	2:	//CleanTip ready?
		IF bStop THEN
			IF fbComplexAction.bBusy THEN
				fbComplexAction.M_Stop();
			ELSE
				nStateAction := 80;
			END_IF
		ELSE
			IF NOT fbComplexAction.bBusy THEN
				A_MoveBack();
				nStateAction := 3;
			END_IF			
		END_IF
		
	3:	//MoveBack
		A_MoveBack();
		IF nStateA_MoveBack >= 80 THEN
			IF nStateA_MoveBack = 99 THEN
				nStateAction := 99;
			ELSE
				nStateAction := 80;
			END_IF
			nStateA_MoveBack := 0;
		END_IF
		
END_CASE
END_ACTION

ACTION A_DilMoveValve:
stError.POUState := nStateAction;

CASE nStateAction OF
	0:	
		IF bStop THEN
			nStateAction := 80;
		ELSE
			IF stGCodeRef.pCurrentTool = 0 THEN
				stError.ErrorId := E_ErrorIdGCode.ERRORID_NoSelectedTool;
				nStateAction := 99;
			ELSE
				IF NOT fbItpReadRParams.bBusy THEN
					MEMSET(ADR(stActionData),0,SIZEOF(stActionData));
					stActionData.eAction := E_Action.ACTION_DilMoveValve;
					stActionData.aParams[1] := LREAL_TO_DINT(alrRParam[1]); //ValvePos
					stError.ErrorId := stGCodeRef.pCurrentTool^.M_ExeAction(stActionData);
					IF stError.ErrorId > 0 THEN
						nStateAction := 99;
					ELSE
						nStateAction := 1;	
					END_IF
				END_IF
			END_IF
		END_IF
		
	1:	//Ready?
		IF bStop THEN
			stGCodeRef.pCurrentTool^.M_CancelAction(E_Action.ACTION_DilMoveValve);
		END_IF
		
		IF NOT stGCodeRef.pCurrentTool^.P_bBusy THEN
			IF stGCodeRef.pCurrentTool^.P_bError THEN
				stError.ErrorId := stGCodeRef.pCurrentTool^.P_nErrorId;
				nStateAction := 99;
			ELSE
				nStateAction := 80;	
			END_IF
		END_IF
END_CASE
END_ACTION

ACTION A_Dispense:
stError.POUState := nStateAction;

CASE nStateAction OF
	0:	//Diluter in Ausgangsposition fahren (BOTTOM)	
		IF bStop THEN
			nStateAction := 80;
		ELSE
			IF stGCodeRef.pCurrentTool = 0 THEN
				stError.ErrorId := E_ErrorIdGCode.ERRORID_NoSelectedTool;
				nStateAction := 99;
			ELSE 
				IF stGCodeRef.pCurrentTool^.P_eObjectType = E_ObjectType.OBJECTTYPE_PassivPip THEN
					pPassivPip := stGCodeRef.pCurrentTool;
				ELSE
					nStateAction := 99;
					RETURN;
				END_IF
				
				IF NOT fbItpReadRParams.bBusy THEN
					MEMSET(ADR(stActionData),0,SIZEOF(stActionData));
					stActionData.eAction := E_Action.ACTION_DilMovePlunger;
					stActionData.aParams[1] := 24000;
					stActionData.aParams[2] := pPassivPip^.P_pDiluter^.P_nConfigReloadSpeed;
					stActionData.aParams[3] := pPassivPip^.P_pDiluter^.P_nValvePosInput;
					stError.ErrorId := pPassivPip^.P_pDiluter^.M_ExeAction(stActionData);
					IF stError.ErrorId > 0 THEN
						nStateAction := 99;
					ELSE
						nStateAction := 1;
					END_IF
				END_IF
			END_IF
		END_IF
		
	1:	//Diluter ready -> Dispensen + Timer für Startbreak starten 
		IF bStop THEN
			pPassivPip^.P_pDiluter^.M_CancelAction(ACTION_DilMovePlunger);
			nStateAction := 80;
		ELSE
			IF NOT pPassivPip^.P_pDiluter^.M_GetActionBusy(ACTION_DilMovePlunger) THEN
				MEMSET(ADR(stActionData),0,SIZEOF(stActionData));
				stActionData.eAction := E_Action.ACTION_Dispense;
				IF alrRParam[1] > 0.0 THEN
					stActionData.aParams[1] := LREAL_TO_DINT(alrRParam[1]); //Quantity
					nStateAction := 3;
				ELSE
					//Es wird mit max. 2 x Spritzen-Volumen dispenst
					stActionData.aParams[1] := pPassivPip^.P_pDiluter^.P_nSyringeSize * 20;
					tDelay := LREAL_TO_TIME(alrRParam[3]);
					IF tDelay > T#0S THEN	//Delay
						timer(IN:=TRUE,PT:=tDelay);	//Timer starten
						stGCodeRef.aToolTable[stGCodeRef.sNciToPlc.Tool].tDelayStart := tDelay;
						nStateAction := 2;
					ELSE
						stGCodeRef.aToolTable[stGCodeRef.sNciToPlc.Tool].tDelayStart := T#0s;
						nStateAction := 80;
					END_IF					
				END_IF
				stActionData.aParams[2] := LREAL_TO_DINT(alrRParam[2]); //Flow
				stError.ErrorId := stGCodeRef.pCurrentTool^.M_ExeAction(stActionData);
				IF stError.ErrorId > 0 THEN
					nStateAction := 99;
				END_IF
			END_IF
		END_IF
		
	2:	//Warten auf Timer
		IF bStop THEN
			timer(IN:= FALSE);
			stGCodeRef.pCurrentTool^.M_CancelAction(E_Action.ACTION_Dispense);
			nStateAction := 80;
			RETURN;
		END_IF
		timer();
		IF timer.Q THEN
			timer(IN:= FALSE);		
			nStateAction := 80;
		END_IF
	
	3:	//Warten bis Dispensen fertig
		IF bStop THEN
			pPassivPip^.M_CancelAction(E_Action.ACTION_Dispense);
			nStateAction := 80;
		ELSE
			IF NOT pPassivPip^.M_GetActionBusy(E_Action.ACTION_Dispense) THEN
				nStateAction := 80;
			END_IF
		END_IF
END_CASE
END_ACTION

ACTION A_DispenseDrops:
stError.POUState := nStateAction;

CASE nStateAction OF
	0:	
		IF bStop THEN
			nStateAction := 80;
		ELSE
			IF stGCodeRef.pCurrentTool = 0 THEN
				stError.ErrorId := E_ErrorIdGCode.ERRORID_NoSelectedTool;
				nStateAction := 99;
			ELSE
				IF NOT fbItpReadRParams.bBusy THEN
					stGCodeRef.aToolTable[stGCodeRef.sNciToPlc.Tool].bIsInAction1 := FALSE;
					MEMSET(ADR(stActionData),0,SIZEOF(stActionData));
					stActionData.eAction := E_Action.ACTION_DispenseDrops;
					stActionData.aParams[1] := LREAL_TO_DINT(alrRParam[1]); //Drops
					stActionData.aParams[2] := 1;
					stActionData.aParams[4] := LREAL_TO_DINT(alrRParam[3]); //Drops für Slave bei TwinPip 
					stError.ErrorId := stGCodeRef.pCurrentTool^.M_ExeAction(stActionData);
					IF stError.ErrorId > 0 THEN
						nStateAction := 99;
					ELSE
						IF stActionData.aParams[1] = 0 THEN //Dauerdispensen
							stGCodeRef.aToolTable[stGCodeRef.sNciToPlc.Tool].bIsInAction1 := TRUE;
							tDelay := LREAL_TO_TIME(alrRParam[2]); //Delay
							IF tDelay > T#0S THEN	//Delay
								timer(IN:=TRUE,PT:=tDelay);	//Timer starten
								stGCodeRef.aToolTable[stGCodeRef.sNciToPlc.Tool].tDelayStart := tDelay;
								nStateAction := 2;								
							ELSE
								stGCodeRef.aToolTable[stGCodeRef.sNciToPlc.Tool].tDelayStart := T#0S;
								nStateAction := 80;
							END_IF
						ELSE
							nStateAction := 1;
						END_IF
					END_IF
				END_IF
			END_IF
		END_IF
		
	1:	//Dispense ready?
		IF bStop THEN
			stGCodeRef.pCurrentTool^.M_CancelAction(E_Action.ACTION_DispenseDrops);
			stGCodeRef.aToolTable[stGCodeRef.sNciToPlc.Tool].bIsInAction1 := FALSE;
		END_IF
		
		IF NOT stGCodeRef.pCurrentTool^.P_bBusy THEN
			stGCodeRef.aToolTable[stGCodeRef.sNciToPlc.Tool].bIsInAction1 := FALSE;
			IF stGCodeRef.pCurrentTool^.P_bError THEN
				stError.ErrorId := stGCodeRef.pCurrentTool^.P_nErrorId;
				nStateAction := 99;
			ELSE
				nStateAction := 80;	
			END_IF
		END_IF
		
	2:	//Warten auf Timer
		IF bStop THEN
			timer(IN:= FALSE);
			stGCodeRef.pCurrentTool^.M_CancelAction(E_Action.ACTION_DispenseDrops);
			stGCodeRef.aToolTable[stGCodeRef.sNciToPlc.Tool].bIsInAction1 := FALSE;
			nStateAction := 80;
			RETURN;
		END_IF
		timer();
		IF timer.Q THEN
			timer(IN:= FALSE);		
			nStateAction := 80;
		END_IF		
END_CASE
END_ACTION

ACTION A_Expose:
stError.POUState := nStateAction;

CASE nStateAction OF
	0:	
		IF bStop THEN
			nStateAction := 80;
		ELSE
			IF stGCodeRef.pCurrentTool = 0 THEN
				stError.ErrorId := E_ErrorIdGCode.ERRORID_NoSelectedTool;
				nStateAction := 99;
			ELSE
				IF NOT fbItpReadRParams.bBusy THEN
					MEMSET(ADR(stActionData),0,SIZEOF(stActionData));
					stActionData.eAction := E_Action.ACTION_Expose;
					stActionData.aParams[1] := LREAL_TO_DINT(alrRParam[1]); //Ctrl
					stActionData.aParams[2] := LREAL_TO_DINT(alrRParam[2]); //Brightness
					stActionData.aParams[3] := LREAL_TO_DINT(alrRParam[3]); //Time
					stError.ErrorId := stGCodeRef.pCurrentTool^.M_ExeAction(stActionData);
					IF stError.ErrorId > 0 THEN
						nStateAction := 99;
					ELSE
						IF stActionData.aParams[3] = 0 THEN
							nStateAction := 80;
						ELSE
							nStateAction := 1;	
						END_IF
					END_IF
				END_IF
			END_IF
		END_IF
		
	1:	//Expose ready?
		IF bStop THEN
			stGCodeRef.pCurrentTool^.M_CancelAction(E_Action.ACTION_Expose);
		END_IF
		
		IF NOT stGCodeRef.pCurrentTool^.P_bBusy THEN
			IF stGCodeRef.pCurrentTool^.P_bError THEN
				stError.ErrorId := stGCodeRef.pCurrentTool^.P_nErrorId;
				nStateAction := 99;
			ELSE
				nStateAction := 80;	
			END_IF
		END_IF
END_CASE
END_ACTION

ACTION A_Extrude:
stError.POUState := nStateAction;
CASE nStateAction OF
	0:	
		IF bStop THEN
			nStateAction := 80;
		ELSE
			IF stGCodeRef.pCurrentTool = 0 THEN
				stError.ErrorId := E_ErrorIdGCode.ERRORID_NoSelectedTool;
				nStateAction := 99;
			ELSE
				IF NOT fbItpReadRParams.bBusy THEN
					//Falls Extruder noch nicht ready, weil er z.B. noch in Decomp-Phase ist, warten!
					IF stGCodeRef.pCurrentTool^.M_GetActionBusy(E_Action.ACTION_Extrude) THEN
						RETURN;
					END_IF
					MEMSET(ADR(stActionData),0,SIZEOF(stActionData));
					stActionData.eAction := E_Action.ACTION_Extrude;
					stActionData.aParams[1] := 0;
					stActionData.aParams[2] := 1; //On
					stError.ErrorId := stGCodeRef.pCurrentTool^.M_ExeAction(stActionData);
					IF stError.ErrorId > 0 THEN
						nStateAction := 99;
					ELSE
						stGCodeRef.aToolTable[stGCodeRef.sNciToPlc.Tool].bIsInAction1 := TRUE;
						tDelay := LREAL_TO_TIME(alrRParam[1]); //Delay (Startbreak)
						IF tDelay > T#0S THEN	//Delay
							timer(IN:=TRUE,PT:=tDelay);	//Timer starten
							stGCodeRef.aToolTable[stGCodeRef.sNciToPlc.Tool].tDelayStart := tDelay;
							nStateAction := 1;								
						ELSE
							stGCodeRef.aToolTable[stGCodeRef.sNciToPlc.Tool].tDelayStart := T#0S;
							nStateAction := 80;
						END_IF
					END_IF
				END_IF
			END_IF
		END_IF
		
	1: //Warten auf Timer
		IF bStop THEN
			timer(IN:= FALSE);
			stGCodeRef.pCurrentTool^.M_CancelAction(E_Action.ACTION_Extrude);
			nStateAction := 80;
			RETURN;
		END_IF
		timer();
		IF timer.Q THEN
			timer(IN:= FALSE);
			nStateAction := 80;
		END_IF
END_CASE
END_ACTION

ACTION A_MeasureTool:
stError.POUState := nStateAction;

IF fbComplexAction.bError THEN
	stError.ErrorId :=fbComplexAction.nErrorId;
	nStateAction := 99;
END_IF

CASE nStateAction OF
	0:	//Aktuelles Tool ausgewählt?
		IF stGCodeRef.pCurrentTool = 0 THEN
			stError.Cmd := E_Action.ACTION_MeasureTool;
			stError.ErrorId := E_ErrorIdGCode.ERRORID_NoSelectedTool;
			nStateAction := 99;
		ELSE
			IF NOT fbItpReadRParams.bBusy THEN
				IF fbObjectDirectory.M_GetObjType(LREAL_TO_UINT(alrRParam[1])) = E_ObjectType.OBJECTTYPE_TipCalibrator THEN
					pTarget := fbObjectDirectory.M_GetObjPointer(LREAL_TO_UINT(alrRParam[1]));
					//NCI-Gruppe auflösen
					fbClearGroup(stGCodeRef:= stGCodeRef, bReGearInSlave:= TRUE, bExecute:= TRUE);
					IF NOT fbClearGroup.bBusy THEN
						IF fbClearGroup.bError THEN
							nStateAction := 99;
							stError.ErrorId := fbClearGroup.nErrorId;
						ELSE
							stCurrentPos := pNewTool^.P_stCurrentPosTotal;
							IF bStop THEN
								nStateAction := 80;
							ELSE
								nStateAction := 1;	
							END_IF
						END_IF
						fbClearGroup(stGCodeRef:= stGCodeRef, bExecute:= FALSE);			
					END_IF
				ELSE
					stError.Cmd := E_Action.ACTION_MeasureTool;
					stError.ObjectId := LREAL_TO_UINT(alrRParam[1]);
					stError.ErrorId := E_ErrorIdCmd.ERRORID_UnsuitableTarget;
					nStateAction := 99;
				END_IF
			END_IF
		END_IF

	1:	//Action "MeasureTool" ausführen
		stMeasToolOldOffset := stGCodeRef.pCurrentTool^.P_stAbsPosTotal;
		MEMSET(ADR(stActionData),0,SIZEOF(stActionData));
		stActionData.eAction := E_Action.ACTION_MeasureTool;
		stActionData.nObject := stGCodeRef.pCurrentTool^.P_nObjectID;
		stActionData.nTarget := pTarget^.P_nObjectID;
		stActionData.aParams[2] := LREAL_TO_DINT(alrRParam[3]);

		stError.ErrorId := fbComplexAction.M_ExeAction(stActionData);
		IF stError.ErrorId > 0 THEN
			nStateAction := 99;
		ELSE
			nStateAction := 2;	
		END_IF
		
	2:	//MeasureTool ready? -> Nullpunkt um neuen Offset verschieben
		IF NOT fbComplexAction.bBusy THEN
			stMeasToolNewOffset := stGCodeRef.pCurrentTool^.P_stAbsPosTotal;
			stGCodeRef.sZeroShiftDesc.fShiftX := stGCodeRef.sZeroShiftDesc.fShiftX + stMeasToolOldOffset.X / 1000 -  stMeasToolNewOffset.X / 1000;
			stGCodeRef.sZeroShiftDesc.fShiftY := stGCodeRef.sZeroShiftDesc.fShiftY + stMeasToolOldOffset.Y / 1000 -  stMeasToolNewOffset.Y / 1000;
			stCurrentPos := stGCodeRef.pCurrentTool^.P_stCurrentPosTotal;
			nStateAction := 3;
		END_IF

	3:	//neuen Offset schreiben
		fbItpWriteZeroShiftEx(bExecute:= TRUE, sNciToPlc:= stGCodeRef.sNciToPlc, nZsNo:= 54, sZeroShiftDesc:= stGCodeRef.sZeroShiftDesc);
		IF NOT fbItpWriteZeroShiftEx.bBusy THEN
			IF fbItpWriteZeroShiftEx.bErr THEN
				stError.ErrorId := UDINT_TO_UINT(fbItpWriteZeroShiftEx.nErrId);
				nStateAction := 99;
			ELSE
				A_MoveBack();
				nStateAction := 4;
			END_IF
			fbItpWriteZeroShiftEx(bExecute:= FALSE, sNciToPlc:= stGCodeRef.sNciToPlc, sZeroShiftDesc:= stGCodeRef.sZeroShiftDesc);
		END_IF
		
	4:	//MoveBack
		A_MoveBack();
		IF nStateA_MoveBack >= 80 THEN
			IF nStateA_MoveBack = 99 THEN
				nStateAction := 99;
			ELSE
				nStateAction := 80;
			END_IF
			nStateA_MoveBack := 0;
		END_IF
END_CASE
END_ACTION

ACTION A_MoveBack:
CASE nStateA_MoveBack OF
	0:	//MoveXY Ausgangspunkt (stCurrentPos)
		MEMSET(ADR(stActionData),0,SIZEOF(stActionData));
		stActionData.eAction := E_Action.ACTION_MoveXY;
		stActionData.aParams[1] := E_MoveMode.MODE_AbsWithOffset;
		stActionData.aParams[2] := REAL_TO_DINT(stCurrentPos.X);
		stActionData.aParams[3] := REAL_TO_DINT(stCurrentPos.Y);
		stActionData.aParams[4] := -1; //max Speed X
		stActionData.aParams[5] := -1; //max Speed Y
		stError.ErrorId := stGCodeRef.pCurrentTool^.M_ExeAction(stActionData);
		IF stError.ErrorId > 0 THEN
			nStateA_MoveBack := 99;
		ELSE
			nStateA_MoveBack := 1;
		END_IF
	
	1:	//MoveXY ready? -> MoveZ Ausgangspunkt (stCurrentPos)
		IF NOT stGCodeRef.pCurrentTool^.M_GetActionBusy(E_Action.ACTION_MoveXY) THEN
			IF stGCodeRef.pCurrentTool^.P_eObjectType = E_ObjectType.OBJECTTYPE_TwinPiezoHolder THEN
				//Einschwenken, falls ausgeschwenkt
				pTwinPiezoHolder := stGCodeRef.pCurrentTool;
				IF pTwinPiezoHolder^.P_eCurrentSwivelState = E_SwivelState.Original THEN
					MEMSET(ADR(stActionData),0,SIZEOF(stActionData));
					stActionData.eAction := E_Action.ACTION_Swivel;
					stActionData.aParams[1] := 1;
					stError.ErrorId := pTwinPiezoHolder^.M_ExeAction(stActionData);
					IF stError.ErrorId > 0 THEN
						nStateA_MoveBack := 99;
					ELSE
						nStateA_MoveBack := 2;
					END_IF
				ELSE
					nStateA_MoveBack := 3;		
				END_IF
			ELSE
				nStateA_MoveBack := 3;	
			END_IF
		END_IF	
	
	2:	//TwinPiezoHolder ready?
		IF NOT stGCodeRef.pCurrentTool^.M_GetActionBusy(E_Action.ACTION_Swivel) THEN
			nStateA_MoveBack := 3;
		END_IF
	
	3:	//NCI-Gruppe wieder erstellen
		fbBuildGroup(stGCodeRef:= stGCodeRef, bExecute:= TRUE);
		IF NOT fbBuildGroup.bBusy THEN
			IF fbBuildGroup.bError THEN
				stError.ErrorId := fbBuildGroup.nErrorId;
				nStateA_MoveBack := 99;
			ELSE
				nStateA_MoveBack := 80;
			END_IF
			fbBuildGroup(stGCodeRef:= stGCodeRef, bExecute:= FALSE);
		END_IF	
END_CASE
END_ACTION

ACTION A_MoveFree:
CASE nStateA_MoveFree OF
	0:	
		MEMSET(ADR(stActionData),0,SIZEOF(stActionData));
		stActionData.eAction := E_Action.ACTION_MoveZ;
		stActionData.aParams[1] := E_MoveMode.MODE_Free;
		stActionData.aParams[3] := -1;

		stError.ErrorId := stGCodeRef.pCurrentTool^.M_ExeAction(stActionData);
		IF stError.ErrorId > 0 THEN
			nStateA_MoveFree := 99;
		ELSE
			nStateA_MoveFree := 1;
		END_IF
	
	1:	//MoveXY ready? -> MoveZ Ausgangspunkt (stCurrentPos)
		IF NOT stGCodeRef.pCurrentTool^.M_GetActionBusy(E_Action.ACTION_MoveZ) THEN
			nStateA_MoveFree := 2;
		END_IF	
	
	2:	//NCI-Gruppe wieder erstellen
		fbBuildGroup(stGCodeRef:= stGCodeRef, bExecute:= TRUE);
		IF NOT fbBuildGroup.bBusy THEN
			IF fbBuildGroup.bError THEN
				stError.ErrorId := fbBuildGroup.nErrorId;
				nStateA_MoveFree := 99;
			ELSE
				nStateA_MoveFree := 80;
			END_IF
			fbBuildGroup(stGCodeRef:= stGCodeRef, bExecute:= FALSE);
		END_IF	
END_CASE
END_ACTION

ACTION A_MoveZHome:
stError.POUState := nStateAction;

IF stGCodeRef.pCurrentTool^.P_bError THEN
	stError.ErrorId := stGCodeRef.pCurrentTool^.P_nErrorId;
	nStateAction := 99;
END_IF

CASE nStateAction OF
	0:	//Aktuelles Tool ausgewählt?
		IF stGCodeRef.pCurrentTool = 0 THEN
			stError.ErrorId := E_ErrorIdGCode.ERRORID_NoSelectedTool;
			nStateAction := 99;
		ELSE //Interpolationsgruppe auflösen (notwendig für Step3)
			fbClearGroup(stGCodeRef:= stGCodeRef,bReGearInSlave:= TRUE, bExecute:= TRUE);
			IF NOT fbClearGroup.bBusy THEN
				IF fbClearGroup.bError THEN
					nStateAction := 99;
					stError.ErrorId := fbClearGroup.nErrorId;
				ELSE
					stCurrentPos := pNewTool^.P_stCurrentPosTotal;
					IF bStop THEN
						nStateAction := 80;
					ELSE
						nStateAction := 1;	
					END_IF
				END_IF
				fbClearGroup(stGCodeRef:= stGCodeRef, bExecute:= FALSE);
			END_IF
		END_IF
		
	1:	//MoveZ
		IF bStop THEN
			nStateAction := 80;
		ELSE
			MEMSET(ADR(stActionData),0,SIZEOF(stActionData));
			stActionData.eAction := E_Action.ACTION_MoveZ;
			stActionData.aParams[1] := E_MoveMode.MODE_Home;
			stActionData.aParams[3]  := -1; //MaxSpeed
			stError.ErrorId := stGCodeRef.pCurrentTool^.M_ExeAction(stActionData);
			IF stError.ErrorId > 0 THEN
				nStateAction := 99;
			ELSE
				nStateAction := 2;
			END_IF
		END_IF
		
	2:	//MoveZ ready? -> aktuelle Position auf Q1-Achse übertragen
		IF NOT stGCodeRef.pCurrentTool^.M_GetActionBusy(E_Action.ACTION_MoveZ) THEN
			stCurrentPos := stGCodeRef.pCurrentTool^.P_stCurrentPosTotal;
 			fbMcSetPosition(Axis:= AxisRefQ1, Execute:= TRUE, Position:= stCurrentPos.Z / 1000.0 - stGCodeRef.sZeroShiftDesc.fShiftZ , Options:= sSetPositionOptions);
			nStateAction := 3;	
		END_IF
		
	3:	//SetPosition ready?
		fbMcSetPosition(Axis:= AxisRefQ1);
		IF NOT fbMcSetPosition.Busy THEN
			IF fbMcSetPosition.Error THEN
				stError.ErrorId := UDINT_TO_UINT(fbMcSetPosition.ErrorID);
				nStateAction := 99;
			ELSE
				IF bStop THEN
					nStateAction := 80;
				ELSE
					nStateAction := 4;	
				END_IF
			END_IF
			fbMcSetPosition(Axis:= AxisRefQ1 , Execute:= FALSE);
		END_IF
		
	4:	//Interpolationsgruppe bilden
		fbBuildGroup(stGCodeRef:= stGCodeRef, bExecute:= TRUE);
		IF NOT fbBuildGroup.bBusy THEN
			IF fbBuildGroup.bError THEN
				stError.ErrorId := fbBuildGroup.nErrorId;
				nStateAction := 99;
			ELSE
				nStateAction := 80;
			END_IF
			fbBuildGroup(stGCodeRef:= stGCodeRef, bExecute:= FALSE);
		END_IF
END_CASE
END_ACTION

ACTION A_PipPostSequence:
stError.POUState := nStateAction;

IF fbComplexAction.bError THEN
	stError.ErrorId :=fbComplexAction.nErrorId;
	nStateAction := 99;
	RETURN;
END_IF

CASE nStateAction OF
	0:	//R-Parameter auswerten und validieren
		IF stGCodeRef.pCurrentTool = 0 THEN
			stError.ErrorId := E_ErrorIdGCode.ERRORID_NoSelectedTool;
			nStateAction := 99;
		ELSE
			IF NOT fbItpReadRParams.bBusy THEN
				//alle Paramter validieren und TargetIds zwischenspeichern
				nTgtNrStrob := LREAL_TO_UINT(alrRParam[1]);
				nDispenseTest := LREAL_TO_DINT(alrRParam[2]);
				
				nTgtNrWS_DispenseWaste1	:= LREAL_TO_UINT(alrRParam[3]);
				nSpecPointNr_DispenseWaste1 := LREAL_TO_UINT(alrRParam[4]);
				nQuantity_DispenseWaste1 := LREAL_TO_DINT(alrRParam[5]);
				nFlow_DispenseWaste1 := LREAL_TO_DINT(alrRParam[6]);
				
				nTgtNrSource := LREAL_TO_UINT(alrRParam[7]);
				nGetSampleColSlotNr := LREAL_TO_DINT(alrRParam[8]);
				nGetSampleRow := LREAL_TO_DINT(alrRParam[9]);
				nGetSampleQuantity := LREAL_TO_DINT(alrRParam[10]);
				nGetSampleFlow := LREAL_TO_DINT(alrRParam[11]);
				nGetSampleDelay := LREAL_TO_DINT(alrRParam[12]);
				
				nTgtNrWS_DispenseWaste2 := LREAL_TO_UINT(alrRParam[13]);
				nSpecPointNr_DispenseWaste2 := LREAL_TO_UINT(alrRParam[14]);
				nQuantity_DispenseWaste2 := LREAL_TO_DINT(alrRParam[15]);
				nFlow_DispenseWaste2 := LREAL_TO_DINT(alrRParam[16]);
				
				nTgtNrWS_Wash1 := LREAL_TO_UINT(alrRParam[17]);
				nSpecPointNr_Wash1 := LREAL_TO_UINT(alrRParam[18]);
				nWashFlow_Wash1 := LREAL_TO_DINT(alrRParam[19]);
				nWashTime_Wash1 := LREAL_TO_DINT(alrRParam[20]);

				nTgtNrWS_Wash2 := LREAL_TO_UINT(alrRParam[21]);
				nSpecPointNr_Wash2 := LREAL_TO_UINT(alrRParam[22]);
				nWashFlow_Wash2 := LREAL_TO_DINT(alrRParam[23]);
				nWashTime_Wash2 := LREAL_TO_DINT(alrRParam[24]);
				
				nTgtNrDryPad_Dry1 := LREAL_TO_UINT(alrRParam[25]);
				nDryCount_Dry1 := LREAL_TO_USINT(alrRParam[26]);
				nDryTime_Dry1 := LREAL_TO_DINT(alrRParam[27]);
				
				//Check 1. DispenseTest
				IF nDispenseTest > 0 THEN
					IF NOT M_ValidateTargetNr(nTgtNrStrob) THEN
						stError.ErrorId := E_ErrorIdGCode.ERRORID_InvalidRParameter;
						stError.ErrorId2 := 1;
						nStateAction := 99;
						RETURN;
					END_IF
				END_IF
				
				//Check 2. DispenseWaste
				IF nQuantity_DispenseWaste1 > 0 THEN
					IF NOT M_ValidateTargetNr(nTgtNrWS_DispenseWaste1) THEN
						stError.ErrorId := E_ErrorIdGCode.ERRORID_InvalidRParameter;
						stError.ErrorId2 := 3;
						nStateAction := 99;
						RETURN;
					END_IF
					//Flow muss größer 0 sein!
				END_IF
				
				//Check 3. GetPipSample (Waschlösung)
				IF nGetSampleQuantity > 0 THEN //wenn 0, dann werden die nächsten beiden Schritte auch ausgelassen und müssen nicht gecheckt werden
					IF M_ValidateTargetNr(nTgtNrSource) THEN
						pTarget := fbObjectDirectory.M_GetObjPointer(stGCodeRef.aTargetTable[nTgtNrSource]);
						IF pTarget = 0 THEN
							stError.ErrorId := E_ErrorIdGCode.ERRORID_InvalidRParameter;
							stError.ErrorId2 := 7;
							nStateAction := 99;
							RETURN;
						END_IF
						IF pTarget^.P_eObjectType = E_ObjectType.OBJECTTYPE_Mtp THEN
							pMtp := pTarget;
							IF NOT(nGetSampleColSlotNr > 0 AND nGetSampleColSlotNr <= pMtp^.P_nCols) THEN
								stError.ErrorId := E_ErrorIdGCode.ERRORID_InvalidRParameter;
								stError.ErrorId2 := 8;
								nStateAction := 99;
								RETURN;
							END_IF
							IF NOT(nGetSampleRow > 0 AND nGetSampleRow <= pMtp^.P_nRows) THEN
								stError.ErrorId := E_ErrorIdGCode.ERRORID_InvalidRParameter;
								stError.ErrorId2 := 9;
								nStateAction := 99;
								RETURN;
							END_IF
						ELSIF pTarget^.P_eObjectType = E_ObjectType.OBJECTTYPE_VialRack THEN
							pVialRack := pTarget;						
							//Im Slot muss auch ein Vial sein!
							pPieceSlot := pVialRack^.M_GetSlot(DINT_TO_UINT(nGetSampleColSlotNr));
							IF pPieceSlot = 0 THEN
								stError.ErrorId := E_ErrorIdGCode.ERRORID_InvalidRParameter;
								stError.ErrorId2 := 8;
								nStateAction := 99;
								RETURN;
							END_IF
							IF pPieceSlot^.P_pPiece = 0 THEN
								stError.ErrorId := E_ErrorIdGCode.ERRORID_InvalidRParameter;
								stError.ErrorId2 := 3;
								nStateAction := 99;
								RETURN;
							END_IF
						END_IF
					ELSE
						stError.ErrorId := E_ErrorIdGCode.ERRORID_InvalidRParameter;
						stError.ErrorId2 := 7;
						nStateAction := 99;
						RETURN;
					END_IF
					
					IF nGetSampleFlow < 1 THEN
						stError.ErrorId := E_ErrorIdGCode.ERRORID_InvalidRParameter;
						stError.ErrorId2 := 11;
						nStateAction := 99;
						RETURN;
					END_IF
					
					//Check 4. DispenseWaste
					IF nQuantity_DispenseWaste2 > 0 THEN
						IF NOT M_ValidateTargetNr(nTgtNrWS_DispenseWaste2) THEN
							stError.ErrorId := E_ErrorIdGCode.ERRORID_InvalidRParameter;
							stError.ErrorId2 := 13;
							nStateAction := 99;
							RETURN;
						END_IF
						
						IF nFlow_DispenseWaste2 = 0 THEN
							stError.ErrorId := E_ErrorIdGCode.ERRORID_InvalidRParameter;
							stError.ErrorId2 := 16;
							nStateAction := 99;
							RETURN;
						END_IF
					END_IF
					//Check 5. WashTool
					IF nWashTime_Wash1 > 0 THEN
						IF NOT M_ValidateTargetNr(nTgtNrWS_Wash1) THEN
							stError.ErrorId := E_ErrorIdGCode.ERRORID_InvalidRParameter;
							stError.ErrorId2 := 17;
							nStateAction := 99;
							RETURN;
						END_IF
						IF nWashFlow_Wash1 = 0 THEN
							stError.ErrorId := E_ErrorIdGCode.ERRORID_InvalidRParameter;
							stError.ErrorId2 := 19;
							nStateAction := 99;
							RETURN;
						END_IF
					END_IF
				END_IF
				
				//Check 6. WashTool
				IF nWashTime_Wash2 > 0 THEN
					IF NOT M_ValidateTargetNr(nTgtNrWS_Wash2) THEN
						stError.ErrorId := E_ErrorIdGCode.ERRORID_InvalidRParameter;
						stError.ErrorId2 := 21;
						nStateAction := 99;
						RETURN;
					END_IF
					IF nWashFlow_Wash2 = 0 THEN
						stError.ErrorId := E_ErrorIdGCode.ERRORID_InvalidRParameter;
						stError.ErrorId2 := 23;
						nStateAction := 99;
						RETURN;
					END_IF
				END_IF
					
				//Check 7. DryPip
				IF nDryCount_Dry1 > 0 THEN
					IF NOT M_ValidateTargetNr(nTgtNrDryPad_Dry1) THEN
						stError.ErrorId := E_ErrorIdGCode.ERRORID_InvalidRParameter;
						stError.ErrorId2 := 25;
						nStateAction := 99;
						RETURN;
					END_IF
				END_IF
				nStateAction := 1;
			END_IF
		END_IF
		
	
	1:	//NCI-Gruppe auflösen
		fbClearGroup(stGCodeRef:= stGCodeRef, bReGearInSlave:= TRUE, bExecute:= TRUE);
		IF NOT fbClearGroup.bBusy THEN
			IF fbClearGroup.bError THEN
				nStateAction := 99;
				stError.ErrorId := fbClearGroup.nErrorId;
			ELSE
				stCurrentPos := pNewTool^.P_stCurrentPosTotal;
				IF bStop THEN
					nStateAction := 80;
				ELSE
					nStateAction := 2;
				END_IF
			END_IF
			fbClearGroup(stGCodeRef:= stGCodeRef, bExecute:= FALSE);			
		END_IF
	
	2:	//DispenseTest start
		IF bStop THEN
			nStateAction := 80;
			RETURN;
		END_IF
		
		IF nDispenseTest > 0 THEN
			MEMSET(ADR(stActionData),0,SIZEOF(stActionData));
			stActionData.eAction := E_Action.ACTION_DispenseTest;
			stActionData.nObject := stGCodeRef.pCurrentTool^.P_nObjectID;
			stActionData.nTarget := stGCodeRef.aTargetTable[nTgtNrStrob];
			stActionData.aParams[1] := nDispenseTest;
			stActionData.aParams[2] := 1; //Inhibit dispense trials
			stError.ErrorId := fbComplexAction.M_ExeAction(stActionData);
			IF stError.ErrorId > 0 THEN
				nStateAction := 99;
			ELSE
				alrRParam[1] := 0.0;
				nStateAction := 3;
			END_IF
		ELSE
			nStateAction := 3;
		END_IF
	
	3:	//DispenseTest ready?
		IF NOT fbComplexAction.bBusy THEN
			IF fbComplexAction.P_bLastActionResult THEN
				alrRParam[1] := DINT_TO_LREAL(fbComplexAction.P_nLastActionResult);
				fbComplexAction.P_bLastActionResult := FALSE;
			END_IF
			//in R-Parameter R140 schreiben
			fbItpWriteRParams(sNciToPlc:= stGCodeRef.sNciToPlc, bExecute:= TRUE, pAddr:= ADR(alrRParam), nIndex:= 140, nCount:= 1);
			IF NOT fbItpWriteRParams.bBusy THEN
				IF fbItpWriteRParams.bErr THEN
					nStateAction := 99;
				ELSE
					nStateAction := 4;
				END_IF
				fbItpWriteRParams(sNciToPlc:= stGCodeRef.sNciToPlc, bExecute:= FALSE);
			END_IF
		END_IF
		
	4:	//DispenseWaste start (WashInside)
		IF bStop THEN
			nStateAction := 80;
			RETURN;
		END_IF
	
		IF nQuantity_DispenseWaste1 > 0 THEN
			MEMSET(ADR(stActionData),0,SIZEOF(stActionData));
			stActionData.eAction := E_Action.ACTION_WashTool;
			stActionData.nObject := stGCodeRef.pCurrentTool^.P_nObjectID;
			stActionData.nTarget := stGCodeRef.aTargetTable[nTgtNrWS_DispenseWaste1];
			stActionData.aParams[1] := nSpecPointNr_DispenseWaste1;
			stActionData.aParams[2] := E_WashMode.MODE_WashInside;
			stActionData.aParams[3] := nQuantity_DispenseWaste1;
			stActionData.aParams[4] := nFlow_DispenseWaste1;
			stError.ErrorId := fbComplexAction.M_ExeAction(stActionData);
			IF stError.ErrorId > 0 THEN
				nStateAction := 99;
			ELSE
				nStateAction := 5;	
			END_IF
		ELSE
			nStateAction := 6;
		END_IF
	
	5:	//DispenseWaste ready?
		IF NOT fbComplexAction.bBusy THEN
			nStateAction := 6;
		END_IF
	
	6:	//GetPipSample start (Waschlösung)
		IF bStop THEN
			nStateAction := 80;
			RETURN;
		END_IF
		IF nGetSampleQuantity > 0 THEN
			MEMSET(ADR(stActionData),0,SIZEOF(stActionData));
			stActionData.eAction := E_Action.ACTION_GetPipSample;
			stActionData.nObject := stGCodeRef.pCurrentTool^.P_nObjectID;
			stActionData.nTarget := stGCodeRef.aTargetTable[nTgtNrSource];
			stActionData.aParams[1] := nGetSampleColSlotNr;
			stActionData.aParams[2] := nGetSampleRow;
			stActionData.aParams[3] := nGetSampleQuantity;
			stActionData.aParams[4] := nGetSampleFlow;
			stActionData.aParams[5] := nGetSampleDelay;
			//stActionData.aParams[6] := nGetSampleAirGap;
			//stActionData.aParams[7] := nGetSampleDilBypass;
			stActionData.aParams[8] := 1; //aktivate Piezo
			stError.ErrorId := fbComplexAction.M_ExeAction(stActionData);
			IF stError.ErrorId > 0 THEN
				nStateAction := 99;
			ELSE
				nStateAction := 7;
			END_IF
		
		ELSE
			nStateAction := 12;
		END_IF

	7:	//GetPipSample ready?
		IF NOT fbComplexAction.bBusy THEN
			nStateAction := 8; //DispenseWaste
		END_IF
	8:	//DispenseWaste start (WashInside)
		IF bStop THEN
			nStateAction := 80;
			RETURN;
		END_IF
		
		IF nQuantity_DispenseWaste2 > 0 THEN
			MEMSET(ADR(stActionData),0,SIZEOF(stActionData));
			stActionData.eAction := E_Action.ACTION_WashTool;
			stActionData.nObject := stGCodeRef.pCurrentTool^.P_nObjectID;
			stActionData.nTarget := stGCodeRef.aTargetTable[nTgtNrWS_DispenseWaste2];
			stActionData.aParams[1] := nSpecPointNr_DispenseWaste2;
			stActionData.aParams[2] := E_WashMode.MODE_WashInside;
			stActionData.aParams[3] := nQuantity_DispenseWaste2;
			stActionData.aParams[4] := nFlow_DispenseWaste2;
			stError.ErrorId := fbComplexAction.M_ExeAction(stActionData);
			IF stError.ErrorId > 0 THEN
				nStateAction := 99;
			ELSE
				nStateAction := 9;
			END_IF
		ELSE
			nStateAction := 10;
		END_IF	
		
	9:	//DispenseWaste ready?
		IF NOT fbComplexAction.bBusy THEN
			nStateAction := 10;
		END_IF
	10:	//WashTool(1) start
		IF bStop THEN
			nStateAction := 80;
			RETURN;
		END_IF
		
		IF nWashTime_Wash1 > 0 THEN
			MEMSET(ADR(stActionData),0,SIZEOF(stActionData));
			stActionData.eAction := E_Action.ACTION_WashTool;
			stActionData.nObject := stGCodeRef.pCurrentTool^.P_nObjectID;
			stActionData.nTarget := stGCodeRef.aTargetTable[nTgtNrWS_Wash1];
			stActionData.aParams[1] := nSpecPointNr_Wash1;
			stActionData.aParams[2] := E_WashMode.MODE_WashInOutside;
			stActionData.aParams[3] := 0; //wenn Quantity 0 dann wird nach Time dispenst?
			stActionData.aParams[4] := nWashFlow_Wash1;
			stActionData.aParams[5] := nWashTime_Wash1;
			stError.ErrorId := fbComplexAction.M_ExeAction(stActionData);
			IF stError.ErrorId > 0 THEN
				nStateAction := 99;
			ELSE
				nStateAction := 11;
			END_IF
		ELSE
			nStateAction := 12;
		END_IF
	11:	//WashTool(1) ready?
		IF NOT fbComplexAction.bBusy THEN
			nStateAction := 12;
		END_IF		

	12:	//WashTool(2) start
		IF bStop THEN
			nStateAction := 80;
			RETURN;
		END_IF
		
		IF nWashTime_Wash2 > 0 THEN
			MEMSET(ADR(stActionData),0,SIZEOF(stActionData));
			stActionData.eAction := E_Action.ACTION_WashTool;
			stActionData.nObject := stGCodeRef.pCurrentTool^.P_nObjectID;
			stActionData.nTarget := stGCodeRef.aTargetTable[nTgtNrWS_Wash2];
			stActionData.aParams[1] := nSpecPointNr_Wash2;
			stActionData.aParams[2] := E_WashMode.MODE_WashInOutside;
			stActionData.aParams[3] := 0; //wenn Quantity 0 dann wird nach Time dispenst?
			stActionData.aParams[4] := nWashFlow_Wash2;
			stActionData.aParams[5] := nWashTime_Wash2;
			stError.ErrorId := fbComplexAction.M_ExeAction(stActionData);
			IF stError.ErrorId > 0 THEN
				nStateAction := 99;
			ELSE
				nStateAction := 13;
			END_IF
		ELSE
			nStateAction := 14;
		END_IF
	13:	//WashTool(2) ready?
		IF NOT fbComplexAction.bBusy THEN
			nStateAction := 14;
		END_IF		
		
	14:	//DryPip
		IF bStop THEN
			nStateAction := 80;
			RETURN;
		END_IF
	
		IF nDryCount_Dry1 > 0 THEN
			MEMSET(ADR(stActionData),0,SIZEOF(stActionData));
			stActionData.eAction := E_Action.ACTION_DryPip;
			stActionData.nObject := stGCodeRef.pCurrentTool^.P_nObjectID;
			stActionData.nTarget := stGCodeRef.aTargetTable[nTgtNrDryPad_Dry1];
			stActionData.aParams[1] := nDryTime_Dry1;
			stError.ErrorId := fbComplexAction.M_ExeAction(stActionData);
			IF stError.ErrorId > 0 THEN
				nStateAction := 99;
			ELSE
				nStateAction := 15;	
			END_IF
		ELSE
			nStateAction := 16;
		END_IF
		
	15:	//DryPip ready?
		IF NOT fbComplexAction.bBusy THEN
			nDryCount_Dry1 := nDryCount_Dry1 - 1;
			IF nDryCount_Dry1 > 0 THEN //wiederholen
				nStateAction := 14;
			ELSE
				nStateAction := 16;
			END_IF
		END_IF
		
	16:	//MoveFree
		A_MoveFree();
		IF nStateA_MoveFree >= 80 THEN
			IF nStateA_MoveFree = 99 THEN
				nStateAction := 99;
			ELSE
				nStateAction := 80;
			END_IF
			nStateA_MoveFree := 0;
		END_IF		
	
END_CASE
END_ACTION

ACTION A_PipPreSequence:
stError.POUState := nStateAction;

IF fbComplexAction.bError THEN
	stError.ErrorId :=fbComplexAction.nErrorId;
	nStateAction := 99;
	RETURN;
END_IF

CASE nStateAction OF
	0:	//R-Parameter auswerten und validieren
		IF stGCodeRef.pCurrentTool = 0 THEN
			stError.ErrorId := E_ErrorIdGCode.ERRORID_NoSelectedTool;
			nStateAction := 99;
		ELSE
			IF NOT fbItpReadRParams.bBusy THEN
				//alle Paramter validieren und TargetIds zwischenspeichern
				nTgtNrWS_Wash1 := LREAL_TO_UINT(alrRParam[1]);
				nSpecPointNr_Wash1 := LREAL_TO_UINT(alrRParam[2]);
				nWashFlow_Wash1 := LREAL_TO_DINT(alrRParam[3]);
				nWashTime_Wash1 := LREAL_TO_DINT(alrRParam[4]);
				nTgtNrDryPad_Dry1 := LREAL_TO_UINT(alrRParam[5]);	//kann auch Washstation mit Airblade sein (ab V2.0.8.9)
				nDryCount_Dry1 := LREAL_TO_USINT(alrRParam[6]);		//bei Washstation ist das der SpecPoint der Airblade
				nDryTime_Dry1 := LREAL_TO_DINT(alrRParam[7]);
				nTgtNrSource := LREAL_TO_UINT(alrRParam[8]);
				nGetSampleColSlotNr := LREAL_TO_DINT(alrRParam[9]);
				nGetSampleRow := LREAL_TO_DINT(alrRParam[10]);
				nGetSampleQuantity := LREAL_TO_DINT(alrRParam[11]);
				nGetSampleFlow := LREAL_TO_DINT(alrRParam[12]);
				nGetSampleDelay := LREAL_TO_DINT(alrRParam[13]);
				nGetSampleAirGap := LREAL_TO_DINT(alrRParam[14]);
				nGetSampleDilBypass := LREAL_TO_DINT(alrRParam[15]);
				nTgtNrDryPad_Dry2 := LREAL_TO_UINT(alrRParam[16]);	//kann auch Washstation mit Airblade sein (ab V2.0.8.9)
				nDryCount_Dry2 := LREAL_TO_USINT(alrRParam[17]);	//bei Washstation ist das der SpecPoint der Airblade
				nDryTime_Dry2 := LREAL_TO_DINT(alrRParam[18]);
				nTgtNrStrob := LREAL_TO_UINT(alrRParam[19]);
				nDispenseTest := LREAL_TO_DINT(alrRParam[20]);
				//Check 1. WashTool
				IF nWashTime_Wash1 > 0 THEN
					IF NOT M_ValidateTargetNr(nTgtNrWS_Wash1) THEN
						stError.ErrorId := E_ErrorIdGCode.ERRORID_InvalidRParameter;
						stError.ErrorId2 := 1;
						nStateAction := 99;
						RETURN;
					END_IF
				END_IF
				//Check 2. DryPip
				IF nDryCount_Dry1 > 0 THEN
					IF NOT M_ValidateTargetNr(nTgtNrDryPad_Dry1) THEN
						stError.ErrorId := E_ErrorIdGCode.ERRORID_InvalidRParameter;
						stError.ErrorId2 := 5;
						nStateAction := 99;
						RETURN;
					END_IF
				END_IF
				//Check 3. GetPipSample
				IF nGetSampleQuantity  > 0 THEN
					IF M_ValidateTargetNr(nTgtNrSource) THEN
						pTarget := fbObjectDirectory.M_GetObjPointer(stGCodeRef.aTargetTable[nTgtNrSource]);
						IF pTarget = 0 THEN
							stError.ErrorId := E_ErrorIdGCode.ERRORID_InvalidRParameter;
							stError.ErrorId2 := 8;
							nStateAction := 99;
							RETURN;
						END_IF
						IF pTarget^.P_eObjectType = E_ObjectType.OBJECTTYPE_Mtp THEN
							pMtp := pTarget;
							IF NOT(nGetSampleColSlotNr > 0 AND nGetSampleColSlotNr <= pMtp^.P_nCols) THEN
								stError.ErrorId := E_ErrorIdGCode.ERRORID_InvalidRParameter;
								stError.ErrorId2 := 9;
								nStateAction := 99;
								RETURN;
							END_IF
							IF NOT(nGetSampleRow > 0 AND nGetSampleRow <= pMtp^.P_nRows) THEN
								stError.ErrorId := E_ErrorIdGCode.ERRORID_InvalidRParameter;
								stError.ErrorId2 := 10;
								nStateAction := 99;
								RETURN;
							END_IF
						ELSIF pTarget^.P_eObjectType = E_ObjectType.OBJECTTYPE_VialRack THEN
							pVialRack := pTarget;						
							//Im Slot muss auch ein Vial sein!
							pPieceSlot := pVialRack^.M_GetSlot(DINT_TO_UINT(nGetSampleColSlotNr));
							IF pPieceSlot = 0 THEN
								stError.ErrorId := E_ErrorIdGCode.ERRORID_InvalidRParameter;
								stError.ErrorId2 := 9;
								nStateAction := 99;
								RETURN;
							END_IF
							IF pPieceSlot^.P_pPiece = 0 THEN
								stError.ErrorId := E_ErrorIdGCode.ERRORID_InvalidRParameter;
								stError.ErrorId2 := 9;
								nStateAction := 99;
								RETURN;
							END_IF
						END_IF
					ELSE
						stError.ErrorId := E_ErrorIdGCode.ERRORID_InvalidRParameter;
						stError.ErrorId2 := 8;
						nStateAction := 99;
						RETURN;
					END_IF
					
					IF nGetSampleFlow < 1 THEN
						stError.ErrorId := E_ErrorIdGCode.ERRORID_InvalidRParameter;
						stError.ErrorId2 := 12;
						nStateAction := 99;
						RETURN;
					END_IF
					
					//Check 4. DryPip
					IF nDryCount_Dry2 > 0 THEN
						IF NOT M_ValidateTargetNr(nTgtNrDryPad_Dry2) THEN
							stError.ErrorId := E_ErrorIdGCode.ERRORID_InvalidRParameter;
							stError.ErrorId2 := 16;
							nStateAction := 99;
							RETURN;
						END_IF
					END_IF
					
					IF nDispenseTest > 0 AND NOT M_ValidateTargetNr(nTgtNrStrob) THEN
						stError.ErrorId := E_ErrorIdGCode.ERRORID_InvalidRParameter;
						stError.ErrorId2 := 18;
						nStateAction := 99;
						RETURN;
					END_IF
					
				END_IF
				nStateAction := 1;
			END_IF
		END_IF
		
	1:	//NCI-Gruppe auflösen
		fbClearGroup(stGCodeRef:= stGCodeRef, bReGearInSlave:= TRUE, bExecute:= TRUE);
		IF NOT fbClearGroup.bBusy THEN
			IF fbClearGroup.bError THEN
				nStateAction := 99;
				stError.ErrorId := fbClearGroup.nErrorId;
			ELSE
				stCurrentPos := pNewTool^.P_stCurrentPosTotal;
				IF bStop THEN
					nStateAction := 80;
				ELSE
					nStateAction := 2;
				END_IF
			END_IF
			fbClearGroup(stGCodeRef:= stGCodeRef, bExecute:= FALSE);			
		END_IF
		
	2:	//1. WashTool start
		IF bStop THEN
			nStateAction := 80;
			RETURN;
		END_IF
		
		IF nWashTime_Wash1 > 0 THEN
			MEMSET(ADR(stActionData),0,SIZEOF(stActionData));
			stActionData.eAction := E_Action.ACTION_WashTool;
			stActionData.nObject := stGCodeRef.pCurrentTool^.P_nObjectID;
			stActionData.nTarget := stGCodeRef.aTargetTable[nTgtNrWS_Wash1];
			stActionData.aParams[1] := nSpecPointNr_Wash1;
			stActionData.aParams[2] := E_WashMode.MODE_WashInOutside;
			stActionData.aParams[3] := 0; //wenn Quantity 0 dann wird nach Time dispenst?
			stActionData.aParams[4] := nWashFlow_Wash1;
			stActionData.aParams[5] := nWashTime_Wash1;
			stError.ErrorId := fbComplexAction.M_ExeAction(stActionData);
			IF stError.ErrorId > 0 THEN
				nStateAction := 99;
			ELSE
				nStateAction := 3;	
			END_IF
		ELSE
			nStateAction := 4;
		END_IF
		
	3:	//1. WashTool ready?
		IF NOT fbComplexAction.bBusy THEN
			nStateAction := 4;
		END_IF
		
	4:	//2. DryPip start
		IF bStop THEN
			nStateAction := 80;
			RETURN;
		END_IF
	
		//Ab V2.0.8.9 wird unterschieden, ob auf Drypad oder Washstation mit Airblade getrockent wird.
		IF nDryCount_Dry1 > 0 THEN
			MEMSET(ADR(stActionData),0,SIZEOF(stActionData));
			stActionData.nObject := stGCodeRef.pCurrentTool^.P_nObjectID;
			stActionData.nTarget := stGCodeRef.aTargetTable[nTgtNrDryPad_Dry1];
			
			pTarget := fbObjectDirectory.M_GetObjPointer(stGCodeRef.aTargetTable[nTgtNrDryPad_Dry1]);
			IF pTarget^.P_eObjectType = E_ObjectType.OBJECTTYPE_DryPad THEN
				stActionData.eAction := E_Action.ACTION_DryPip;
				stActionData.aParams[1] := nDryTime_Dry1;
			ELSIF pTarget^.P_eObjectType = E_ObjectType.OBJECTTYPE_WashStation THEN
				stActionData.eAction := E_Action.ACTION_WashTool;
				stActionData.aParams[1] := nDryCount_Dry1; //Specpoint
				stActionData.aParams[2] := E_WashMode.MODE_DryOutside;
				stActionData.aParams[5] := nDryTime_Dry1;
			ELSE
				stError.ErrorId := E_ErrorIdCmd.ERRORID_InvalidTarget;
			END_IF
			
			IF stError.ErrorId > 0 THEN
				nStateAction := 99;
			ELSE
				stError.ErrorId := fbComplexAction.M_ExeAction(stActionData);
				IF stError.ErrorId > 0 THEN
					nStateAction := 99;
				ELSE
					nStateAction := 5;	
				END_IF
			END_IF
		ELSE
			nStateAction := 6; //GetPipSample	
		END_IF
	
	5:	//2. DryPip ready?
		IF NOT fbComplexAction.bBusy THEN
			IF pTarget^.P_eObjectType = E_ObjectType.OBJECTTYPE_DryPad THEN
				nDryCount_Dry1 := nDryCount_Dry1 - 1;
				IF nDryCount_Dry1 > 0 THEN
					nStateAction := 4;
				ELSE
					nStateAction := 6; //GetSample
				END_IF
			ELSE
				nStateAction := 6; //GetSample
			END_IF
		END_IF
		
	6:	//3. GetSample start
		IF bStop THEN
			nStateAction := 80;
			RETURN;
		END_IF
	
		IF nGetSampleQuantity > 0 THEN
			MEMSET(ADR(stActionData),0,SIZEOF(stActionData));
			stActionData.eAction := E_Action.ACTION_GetPipSample;
			stActionData.nObject := stGCodeRef.pCurrentTool^.P_nObjectID;
			stActionData.nTarget := stGCodeRef.aTargetTable[nTgtNrSource];
			stActionData.aParams[1] := nGetSampleColSlotNr;
			stActionData.aParams[2] := nGetSampleRow;
			stActionData.aParams[3] := nGetSampleQuantity;
			stActionData.aParams[4] := nGetSampleFlow;
			stActionData.aParams[5] := nGetSampleDelay;
			stActionData.aParams[6] := nGetSampleAirGap;
			stActionData.aParams[7] := nGetSampleDilBypass;
			stError.ErrorId := fbComplexAction.M_ExeAction(stActionData);
			IF stError.ErrorId > 0 THEN
				nStateAction := 99;
			ELSE
				nStateAction := 7;
			END_IF
		ELSE
			nStateAction := 8; //DryPip zum Zweiten
		END_IF
	
	7:	//3. GetSample ready?
		IF NOT fbComplexAction.bBusy THEN
			nStateAction := 8; //DryPip zum Zweiten
		END_IF
		
	8:	//4. DryPip start
		IF bStop THEN
			nStateAction := 80;
			RETURN;
		END_IF
	
		IF nDryCount_Dry2 > 0 THEN
			MEMSET(ADR(stActionData),0,SIZEOF(stActionData));
			stActionData.nObject := stGCodeRef.pCurrentTool^.P_nObjectID;
			stActionData.nTarget := stGCodeRef.aTargetTable[nTgtNrDryPad_Dry2];
			
			pTarget := fbObjectDirectory.M_GetObjPointer(stGCodeRef.aTargetTable[nTgtNrDryPad_Dry2]);
			IF pTarget^.P_eObjectType = E_ObjectType.OBJECTTYPE_DryPad THEN
				stActionData.eAction := E_Action.ACTION_DryPip;
				stActionData.aParams[1] := nDryTime_Dry2;
			ELSIF pTarget^.P_eObjectType = E_ObjectType.OBJECTTYPE_WashStation THEN
				stActionData.eAction := E_Action.ACTION_WashTool;
				stActionData.aParams[1] := nDryCount_Dry2; //Specpoint
				stActionData.aParams[2] := E_WashMode.MODE_DryOutside;
				stActionData.aParams[5] := nDryTime_Dry2;
			ELSE
				stError.ErrorId := E_ErrorIdCmd.ERRORID_InvalidTarget;
			END_IF
			
			IF stError.ErrorId > 0 THEN
				nStateAction := 99;
			ELSE
				stError.ErrorId := fbComplexAction.M_ExeAction(stActionData);
				IF stError.ErrorId > 0 THEN
					nStateAction := 99;
				ELSE
					nStateAction := 9;
				END_IF
			END_IF
		ELSE
			IF nDispenseTest > 0 THEN
				nStateAction := 10; //DispenseTest
			ELSE
				nStateAction := 12;
			END_IF
		END_IF
	
	9:	//DryPip ready?
		IF NOT fbComplexAction.bBusy THEN
			IF pTarget^.P_eObjectType = E_ObjectType.OBJECTTYPE_DryPad THEN
				nDryCount_Dry2 := nDryCount_Dry2 - 1;
				IF nDryCount_Dry2 > 0 THEN //wiederholen
					nStateAction := 8;
				ELSE
					IF nDispenseTest > 0 THEN
						nStateAction := 10; //DispenseTest
					ELSE
						nStateAction := 12;
					END_IF
				END_IF
			ELSE
				IF nDispenseTest > 0 THEN
					nStateAction := 10; //DispenseTest
				ELSE
					nStateAction := 12;
				END_IF
			END_IF
		END_IF
		
	10:	//DispenseTest start
		IF bStop THEN
			nStateAction := 80;
			RETURN;
		END_IF
	
		MEMSET(ADR(stActionData),0,SIZEOF(stActionData));
		stActionData.eAction := E_Action.ACTION_DispenseTest;
		stActionData.nObject := stGCodeRef.pCurrentTool^.P_nObjectID;
		stActionData.nTarget := stGCodeRef.aTargetTable[nTgtNrStrob];
		stActionData.aParams[1] := nDispenseTest;
		fbComplexAction.P_nDispenseTrials := 0;
		stError.ErrorId := fbComplexAction.M_ExeAction(stActionData);
		IF stError.ErrorId > 0 THEN
			nStateAction := 99;
		ELSE
			alrRParam[1] := 0.0;
			nStateAction := 11;
		END_IF
	
	11:	//DispenseTest ready?
		IF NOT fbComplexAction.bBusy THEN
			IF fbComplexAction.P_bLastActionResult THEN
				alrRParam[1] := DINT_TO_LREAL(fbComplexAction.P_nLastActionResult);
				fbComplexAction.P_bLastActionResult := FALSE;
			END_IF
			//in R-Parameter R140 schreiben
			fbItpWriteRParams(sNciToPlc:= stGCodeRef.sNciToPlc, bExecute:= TRUE, pAddr:= ADR(alrRParam), nIndex:= 140, nCount:= 1);
			IF NOT fbItpWriteRParams.bBusy THEN
				IF fbItpWriteRParams.bErr THEN
					nStateAction := 99;
				ELSE
					nStateAction := 12;	
				END_IF
				fbItpWriteRParams(sNciToPlc:= stGCodeRef.sNciToPlc, bExecute:= FALSE);
			END_IF
		END_IF
		
	12:	//MoveFree
		A_MoveFree();
		IF nStateA_MoveFree >= 80 THEN
			IF nStateA_MoveFree = 99 THEN
				nStateAction := 99;
			ELSE
				nStateAction := 80;
			END_IF
			nStateA_MoveFree := 0;
		END_IF	
END_CASE
END_ACTION

ACTION A_SelectTool:
//+++++++++++++++++++++++++++++++++++++++++++++++++++++++++++++++++++++++++++++++++++++++++++++++++++++++++++++
//Änderung ab V2.0.17!
//Beim Toolwechsel wird nicht mehr der Druck oder der Feed eingestellt.
//Nach einem Toolwechsel sollte daher immer M102 ausgeführt werden
stError.POUState := nStateAction;

CASE nStateAction OF
	0:	
		IF bStop THEN
			nStateAction := 80;
		ELSE
			//Checken, ob Toolnummer (T-Paramter) gültig
			IF NOT (stGCodeRef.sNciToPlc.Tool > 0 AND stGCodeRef.sNciToPlc.Tool <= GCode.cMaxGCodeTools) THEN
				stError.ErrorId := E_ErrorIdGCode.ERRORID_InvalidToolNr;
				nStateAction := 99;
				RETURN;
			ELSE
				//Checken, ob ein gültiges Werkzeug zugeordnet
				IF stGCodeRef.aToolTable[stGCodeRef.sNciToPlc.Tool].pMzTool = 0 OR 
											NOT stGCodeRef.aToolTable[stGCodeRef.sNciToPlc.Tool].bIsUsed THEN
					stError.ErrorId := E_ErrorIdGCode.ERRORID_InvalidToolNr;
					nStateAction := 99;
					RETURN;
				END_IF
			END_IF
			
			pNewTool := stGCodeRef.aToolTable[stGCodeRef.sNciToPlc.Tool].pMzTool;
			
			//Achsen freifahren
			IF pNewTool^.P_bIsMESTool THEN //MES-Tool wird vom Freifahren ausgeschlossen, da Faden abreißen würde
				stError.ErrorId := stGCodeRef.pHead^.M_MoveFree(pNewTool);
			ELSE
				stError.ErrorId := stGCodeRef.pHead^.M_MoveFree(0);	
			END_IF
			
			IF stError.ErrorId > 0 THEN
				nStateAction := 99;
				RETURN;
			END_IF
			nStateAction := 1;
		END_IF
		
	1:	//Achsen ready?
		IF NOT stGCodeRef.pHead^.M_GetActionBusy(E_Action.ACTION_MoveZ) THEN
			nStateAction := 3;
			IF bStop THEN
				nStateAction := 80;
			ELSE
				IF pNewTool^.P_eObjectType = E_ObjectType.OBJECTTYPE_TwinPiezoHolder THEN
					pTwinPiezoHolder := pNewTool;
					IF pTwinPiezoHolder^.P_eCurrentSwivelState <> E_SwivelState.Swiveled THEN
						//Einschwenken
						MEMSET(ADR(stActionData),0,SIZEOF(stActionData));
						stActionData.eAction := E_Action.ACTION_Swivel;
						stActionData.aParams[1] := 1;
						stError.ErrorId := pTwinPiezoHolder^.M_ExeAction(stActionData);
						IF stError.ErrorId > 0 THEN
							nStateAction := 99;
							RETURN;					
						END_IF
						nStateAction := 2;	//warten bis eingeschwenkt
					END_IF
 				END_IF
			END_IF
		END_IF
		
		IF stGCodeRef.pHead^.P_bError THEN
			stError.ErrorId := stGCodeRef.pHead^.P_nErrorId;
			nStateAction := 99;
			RETURN;
		END_IF
	
	2:	//TwinPiezoHolder eingeschwenkt?
		IF bStop THEN
			pNewTool^.M_CancelAction(E_Action.ACTION_Swivel);
			nStateAction := 80;
			RETURN;
		END_IF
		
		IF NOT pNewTool^.M_GetActionBusy(E_Action.ACTION_Swivel) THEN
			nStateAction := 3;
		END_IF
		

		//hier kommt dann noch ein zusätzlicher Offset hinzu, welcher sich aus der zukünftigen Objektvermessung ergibt
	3:	//Neue Nullpunktverschiebeung berechnen (Offset vom aktuellen mit Offset von neuem Tool verrechnen)
		//Es gibt 2 Fälle
		IF stGCodeRef.pCurrentTool = 0 THEN //Es erfolgt die erstmalige Tool-auswahl
			stPos1 := stGCodeRef.pHead^.P_stAbsPosTotal;
		ELSE //Es wurde bereits ein Tool ausgewählt -> es findet ein Toolwechsel statt
			stPos1 := stGCodeRef.pCurrentTool^.P_stAbsPosTotal;
		END_IF
			
		stPos2 := pNewTool^.P_stAbsPosTotal;
		
		stGCodeRef.sZeroShiftDesc.fShiftX := stGCodeRef.sZeroShiftDesc.fShiftX + stPos1.X / 1000.0 -  stPos2.X / 1000.0;
		stGCodeRef.sZeroShiftDesc.fShiftY := stGCodeRef.sZeroShiftDesc.fShiftY + stPos1.Y / 1000.0 -  stPos2.Y / 1000.0;

		stGCodeRef.pCurrentTool := pNewTool;
		
		nStateAction := 4;
	
	4:	//Neue Nullpunktverschiebung schreiben
		fbItpWriteZeroShiftEx(bExecute:= TRUE, sNciToPlc:= stGCodeRef.sNciToPlc, nZsNo:= 54, sZeroShiftDesc:= stGCodeRef.sZeroShiftDesc);	
 		IF NOT fbItpWriteZeroShiftEx.bBusy THEN
			IF fbItpWriteZeroShiftEx.bErr THEN
				nStateAction := 99;
			ELSE
				IF bStop THEN
					nStateAction := 80;
				ELSE
					nStateAction := 5;
				END_IF
			END_IF
			fbItpWriteZeroShiftEx(bExecute:= FALSE, sNciToPlc:= stGCodeRef.sNciToPlc, nZsNo:= 54, sZeroShiftDesc:= stGCodeRef.sZeroShiftDesc);
		END_IF
		
	5:	//NCI-Gruppe auflösen
		fbClearGroup(stGCodeRef:= stGCodeRef, bReGearInSlave:= TRUE, bExecute:= TRUE);
		IF NOT fbClearGroup.bBusy THEN
			IF fbClearGroup.bError THEN
				nStateAction := 99;
				stError.ErrorId := fbClearGroup.nErrorId;
			ELSE
				stCurrentPos := pNewTool^.P_stCurrentPosTotal;
				IF bStop THEN
					nStateAction := 80;
				ELSE
					nStateAction := 6;
				END_IF
				
			END_IF
			fbClearGroup(stGCodeRef:= stGCodeRef, bExecute:= FALSE);
		END_IF
		
	6:	//die aktuelle Position des Tools auf die Q1-Achse übertragen
		fbMcSetPosition(Axis:= AxisRefQ1 , Execute:= TRUE, Position:= stCurrentPos.Z / 1000.0 - stGCodeRef.sZeroShiftDesc.fShiftZ , Options:= sSetPositionOptions);
		IF NOT fbMcSetPosition.Busy THEN
			IF fbMcSetPosition.Error THEN
				nStateAction := 99;
			ELSE
				IF bStop THEN
					nStateAction := 80;
				ELSE
					nStateAction := 7;
				END_IF
			END_IF
			fbMcSetPosition(Axis:= AxisRefQ1 , Execute:= FALSE);
		END_IF
		
	7:	//NCI-Gruppe wieder erstellen
		fbBuildGroup(stGCodeRef:= stGCodeRef, bExecute:= TRUE);
		IF NOT fbBuildGroup.bBusy THEN
			IF fbBuildGroup.bError THEN
				stError.ErrorId := fbBuildGroup.nErrorId;
				nStateAction := 99;
			ELSE
				nStateAction := 80;
			END_IF
			fbBuildGroup(stGCodeRef:= stGCodeRef, bExecute:= FALSE);
		END_IF
END_CASE
END_ACTION

ACTION A_Sequence:
stError.POUState := nStateAction;

IF fbComplexAction.bError THEN
	stError.ErrorId :=fbComplexAction.nErrorId;
	nStateAction := 99;
END_IF

IF nStateAction = 0 THEN
	IF stGCodeRef.pCurrentTool = 0 THEN
		//stError.Cmd := E_Action.ACTION_;;
		stError.ErrorId := E_ErrorIdGCode.ERRORID_NoSelectedTool;
		nStateAction := 99;
	ELSE
		IF NOT fbItpReadRParams.bBusy THEN
			nSequenceNr := LREAL_TO_UINT(alrRParam[1]);
			//SequenceNr 1..5 ?
			IF nSequenceNr >= 1 AND nSequenceNr <= 5 THEN
				pSequence := fbSequenceList.M_Get(stGCodeRef.aSequenceIds[nSequenceNr]);
				//Gültige SubSequence?
				IF pSequence > 0 THEN
					//Sequence schon busy?
					IF NOT((pSequence^.eCurrentState = E_SequenceState.State_Idle) OR (pSequence^.eCurrentState = E_SequenceState.State_Ready)) THEN
						nStateAction := 99;
						stError.ErrorId := E_ErrorIdGCode.ERRORID_InvalidSequenceNr;
						RETURN;
					END_IF
					//Steps vorhanden?
					stError.ErrorId := pSequence^.M_CheckForStart();
					IF stError.ErrorId = 0 THEN
						//NCI-Gruppe auflösen
						fbClearGroup(stGCodeRef:= stGCodeRef, bReGearInSlave:= TRUE, bExecute:= TRUE);
						IF NOT fbClearGroup.bBusy THEN
							IF fbClearGroup.bError THEN
								nStateAction := 99;
								stError.ErrorId := fbClearGroup.nErrorId;
							ELSE
								stCurrentPos := pNewTool^.P_stCurrentPosTotal;
								IF bStop THEN
									nStateAction := 80;
								ELSIF bPause THEN
									nStateAction := 2; //sofort in Pause gehen
								ELSE
									GCode.P_bMoveActionsLocked := FALSE;
									pSequence^.M_Start(0);									
									nStateAction := 3; //perform sequence
								END_IF
							END_IF
							fbClearGroup(stGCodeRef:= stGCodeRef, bExecute:= FALSE);			
						END_IF
					ELSE
						nStateAction := 99;				
					END_IF
				ELSE
					stError.ErrorId := E_ErrorIdCmd.ERRORID_SequenceNotExists;
					nStateAction := 99;
				END_IF				
			ELSE
				stError.ErrorId := E_ErrorIdGCode.ERRORID_InvalidSequenceNr;
				nStateAction := 99;
			END_IF
		END_IF
	END_IF
END_IF

IF nStateAction = 1 THEN //Sequence pausieren
	pSequence^.M_Pause();
	pSequence^();
	IF pSequence^.eCurrentState = E_SequenceState.State_Pause THEN
		nStateAction := 2;
	ELSIF pSequence^.eCurrentState = E_SequenceState.State_Error THEN
		nStateAction := 99;
	ELSIF pSequence^.eCurrentState = E_SequenceState.State_Ready THEN
		pSequence^.M_Reset();
		nStateAction := 80;
		RETURN;
	END_IF
ELSIF nStateAction = 2 THEN //Sequence ist pausiert
	IF bStop THEN
		pSequence^.M_Stop();
		nStateAction := 3;
	ELSIF bPause THEN
		bIsInPause := TRUE;
		RETURN;
	ELSIF bContinue THEN
		IF pSequence^.eCurrentState = E_SequenceState.State_Pause THEN	
			pSequence^.M_Continue();
		ELSIF pSequence^.eCurrentState = E_SequenceState.State_Idle THEN //wurde noch nicht gestartet
			pSequence^.M_Start(0);
		END_IF
		nStateAction := 3;
	END_IF
END_IF

IF nStateAction = 3 THEN //perform sequence , wait for ready
	bIsInPause := FALSE;
	IF bStop THEN
		pSequence^.M_Stop();
	ELSIF bPause THEN
		pSequence^.M_Pause();
		nStateAction := 1;
	END_IF
	pSequence^();
	IF pSequence^.eCurrentState = E_SequenceState.State_Ready THEN
		pSequence^.M_Reset();
		nStateAction := 4;
		GCode.P_bMoveActionsLocked := TRUE;
	ELSIF pSequence^.eCurrentState = E_SequenceState.State_Canceled THEN
		pSequence^.M_Reset();
		nStateAction := 80;
	ELSIF pSequence^.eCurrentState = E_SequenceState.State_Error THEN
		pSequence^.M_Reset();
		nStateAction := 99;
	END_IF
END_IF

IF nStateAction = 4 THEN //MoveBack
	A_MoveBack();
	IF nStateA_MoveBack >= 80 THEN
		IF nStateA_MoveBack = 99 THEN
			nStateAction := 99;
		ELSE
			nStateAction := 80;
		END_IF
		nStateA_MoveBack := 0;
	END_IF	
END_IF
END_ACTION

ACTION A_SetPrintParams:
stError.POUState := nStateAction;

IF nStateAction = 0 THEN
	IF NOT fbItpReadRParams.bBusy THEN
		nToolNr := LREAL_TO_USINT(alrRParam[1]);
		ePrintParamType := LREAL_TO_USINT(alrRParam[2]);
		nPrintParamNumerator := LREAL_TO_USINT(alrRParam[3]);
		nPrintParamValue := LREAL_TO_DINT(alrRParam[4]);
		IF nToolNr = 0 THEN //ausgewähltes Tool benutzen
			pNewTool := stGCodeRef.pCurrentTool;
		ELSIF nToolNr >= 1 AND nToolNr <= GCode.cMaxGCodeTools THEN
			pNewTool := stGCodeRef.aToolTable[nToolNr].pMzTool;
		END_IF
		nStateAction := 1;
		IF pNewTool = 0 THEN
			stError.ErrorId := E_ErrorIdGCode.ERRORID_InvalidToolNr;
			nStateAction := 99;
		END_IF
	END_IF
END_IF

IF nStateAction = 1 THEN
	stMethResult := pNewTool^.M_SetPrintParams(ePrintParamType, nPrintParamNumerator, nPrintParamValue);
	IF NOT stMethResult.bBusy THEN
		IF stMethResult.bError THEN
			stError.ObjectId := pNewTool^.P_nObjectID;
			stError.ErrorId := nErrorId := stMethResult.nErrorId;
			nStateAction := 99;
		ELSE
			nStateAction := 80;
		END_IF
	END_IF	
END_IF
END_ACTION

ACTION A_StirrCartridge:
stError.POUState := nStateAction;

IF nStateAction = 0 THEN
	IF bStop THEN
		nStateAction := 80;
	ELSE
		IF stGCodeRef.pCurrentTool = 0 THEN
			stError.ErrorId := E_ErrorIdGCode.ERRORID_NoSelectedTool;
			nStateAction := 99;
		ELSE
			IF NOT fbItpReadRParams.bBusy THEN
				MEMSET(ADR(stActionData),0,SIZEOF(stActionData));
				stActionData.eAction := E_Action.ACTION_StirrCartridge;
				stActionData.aParams[1] := LREAL_TO_DINT(alrRParam[1]);
				stActionData.aParams[2] := LREAL_TO_DINT(alrRParam[2]);
				stActionData.aParams[3] := LREAL_TO_DINT(alrRParam[3]);
				stActionData.aParams[4] := LREAL_TO_DINT(alrRParam[4]);
				stError.ErrorId := stGCodeRef.pCurrentTool^.M_ExeAction(stActionData);
				IF stError.ErrorId > 0 THEN
					nStateAction := 99;
				ELSE
					nStateAction := 80;
				END_IF
			END_IF
		END_IF
	END_IF
END_IF
END_ACTION

ACTION A_SwitchPress:
stError.POUState := nStateAction;

CASE nStateAction OF
	0:	
		IF bStop THEN
			nStateAction := 80;
		ELSE
			IF stGCodeRef.pCurrentTool = 0 THEN
				stError.ErrorId := E_ErrorIdGCode.ERRORID_NoSelectedTool;
				nStateAction := 99;
			ELSE
				IF NOT (stGCodeRef.pCurrentTool^.P_eObjectType = E_ObjectType.OBJECTTYPE_CartDispenser OR
					stGCodeRef.pCurrentTool^.P_eObjectType = E_ObjectType.OBJECTTYPE_CartDispStirrer OR
					stGCodeRef.pCurrentTool^.P_eObjectType = E_ObjectType.OBJECTTYPE_MultiCartHolder OR
					stGCodeRef.pCurrentTool^.P_eObjectType = E_ObjectType.OBJECTTYPE_DeloDot) THEN
					stError.ErrorId := E_ErrorIdCmd.ERRORID_UnsuitableObject;
					nStateAction := 99;
				ELSE
					IF NOT fbItpReadRParams.bBusy THEN
						nChannel := LREAL_TO_USINT(alrRParam[1]);
						tDelay := LREAL_TO_TIME(alrRParam[2]);
						
						MEMSET(ADR(stActionData),0,SIZEOF(stActionData));
						stActionData.eAction := E_Action.ACTION_SwitchPressure;
						stActionData.aParams[1] := 1; //On
						IF tDelay > T#0S THEN	//Delay
							timer(IN:=TRUE,PT:=tDelay);	//Timer starten
							stGCodeRef.aToolTable[stGCodeRef.sNciToPlc.Tool].tDelayStart := tDelay;
							nStateAction := 1;
						ELSE
							stGCodeRef.aToolTable[stGCodeRef.sNciToPlc.Tool].tDelayStart := T#0s;
							nStateAction := 80;
						END_IF
						
						IF stGCodeRef.pCurrentTool^.P_eObjectType = E_ObjectType.OBJECTTYPE_MultiCartHolder THEN
							pMultiCartHolder := stGCodeRef.pCurrentTool;
							CASE nChannel OF
								1:	
									IF pMultiCartHolder^.P_pCartDispenser1 > 0 THEN
										nErrorId := pMultiCartHolder^.P_pCartDispenser1^.M_ExeAction(stActionData);
										stGCodeRef.aToolTable[stGCodeRef.sNciToPlc.Tool].bIsInAction1 := TRUE;
									ELSE
										stError.ErrorId := E_ErrorIdObjMgmt.ERRORID_InvalidPneuChannel;
									END_IF
 								2:
									IF pMultiCartHolder^.P_pCartDispenser2 > 0 THEN
										nErrorId := pMultiCartHolder^.P_pCartDispenser2^.M_ExeAction(stActionData);
										stGCodeRef.aToolTable[stGCodeRef.sNciToPlc.Tool].bIsInAction2 := TRUE;
									ELSE
										stError.ErrorId := E_ErrorIdObjMgmt.ERRORID_InvalidPneuChannel;
									END_IF
 								3:
									IF pMultiCartHolder^.P_pCartDispenser3 > 0 THEN
										nErrorId := pMultiCartHolder^.P_pCartDispenser3^.M_ExeAction(stActionData);
										stGCodeRef.aToolTable[stGCodeRef.sNciToPlc.Tool].bIsInAction3 := TRUE;
									ELSE
										stError.ErrorId := E_ErrorIdObjMgmt.ERRORID_InvalidPneuChannel;
									END_IF
							END_CASE
						ELSE
							//bei den anderen Tools gibt es nur einen Druckkanal, der geschaltet werden kann
 							nErrorId := stGCodeRef.pCurrentTool^.M_ExeAction(stActionData);
							stGCodeRef.aToolTable[stGCodeRef.sNciToPlc.Tool].bIsInAction1 := TRUE;
						END_IF
						
						IF nErrorId > 0 THEN
							nStateAction := 99;
							stGCodeRef.aToolTable[stGCodeRef.sNciToPlc.Tool].bIsInAction1 := FALSE;
							stGCodeRef.aToolTable[stGCodeRef.sNciToPlc.Tool].bIsInAction2 := FALSE;
							stGCodeRef.aToolTable[stGCodeRef.sNciToPlc.Tool].bIsInAction3 := FALSE;
						END_IF
					END_IF
				END_IF
			END_IF			
		END_IF
	
	1:	//Warten auf Timer
		IF bStop THEN
			timer(IN:= FALSE);
			stActionData.aParams[1] := 0; //off
			stGCodeRef.pCurrentTool^.M_ExeAction(stActionData);
			nStateAction := 80;
			RETURN;
		END_IF
		timer();
		IF timer.Q THEN
			timer(IN:= FALSE);		
			nStateAction := 80;
		END_IF	
END_CASE
		
IF nStateAction = 99 THEN
	timer(IN:= FALSE);
END_IF
END_ACTION

ACTION A_UniDispense:
stError.POUState := nStateAction;

CASE nStateAction OF
	0:	
		IF bStop THEN
			nStateAction := 80;
		ELSE
			IF stGCodeRef.pCurrentTool = 0 THEN
				stError.ErrorId := E_ErrorIdGCode.ERRORID_NoSelectedTool;
				nStateAction := 99;
			ELSE
				IF NOT fbItpReadRParams.bBusy THEN
					stGCodeRef.aToolTable[stGCodeRef.sNciToPlc.Tool].bIsInAction1 := FALSE;
					nUniDispParam1 := LREAL_TO_DINT(alrRParam[2]);
					nUniDispParam2 := LREAL_TO_DINT(alrRParam[3]);
					stError.ErrorId := stGCodeRef.pCurrentTool^.M_StartUniDispense(nParam1:= nUniDispParam1, nParam2:= nUniDispParam2, bIsContinous=> bUnitDispIsContinous); 
					IF stError.ErrorId > 0 THEN
						nStateAction := 99;
					ELSE
						IF bUnitDispIsContinous THEN //Dauerdispensen
							stGCodeRef.aToolTable[stGCodeRef.sNciToPlc.Tool].bIsInAction1 := TRUE;
							tDelay := LREAL_TO_TIME(alrRParam[1]); //Delay
							IF tDelay > T#0S THEN	//Delay
								timer(IN:=TRUE,PT:=tDelay);	//Timer starten
								stGCodeRef.aToolTable[stGCodeRef.sNciToPlc.Tool].tDelayStart := tDelay;
								nStateAction := 2;								
							ELSE
								stGCodeRef.aToolTable[stGCodeRef.sNciToPlc.Tool].tDelayStart := T#0S;
								nStateAction := 80;
							END_IF
						ELSE
							nStateAction := 1;
						END_IF
					END_IF
				END_IF
			END_IF
		END_IF
		
	1:	//Dispense ready?
		IF bStop THEN
			stGCodeRef.pCurrentTool^.M_StopUniDispense();
			stGCodeRef.aToolTable[stGCodeRef.sNciToPlc.Tool].bIsInAction1 := FALSE;
		END_IF
		
		IF NOT stGCodeRef.pCurrentTool^.P_bBusy THEN
			stGCodeRef.aToolTable[stGCodeRef.sNciToPlc.Tool].bIsInAction1 := FALSE;
			IF stGCodeRef.pCurrentTool^.P_bError THEN
				stError.ErrorId := stGCodeRef.pCurrentTool^.P_nErrorId;
				nStateAction := 99;
			ELSE
				nStateAction := 80;	
			END_IF
		END_IF
		
	2:	//Warten auf Timer
		IF bStop THEN
			timer(IN:= FALSE);
			stGCodeRef.pCurrentTool^.M_StopUniDispense();
			stGCodeRef.aToolTable[stGCodeRef.sNciToPlc.Tool].bIsInAction1 := FALSE;
			nStateAction := 80;
			RETURN;
		END_IF
		timer();
		IF timer.Q THEN
			timer(IN:= FALSE);		
			nStateAction := 80;
		END_IF		
END_CASE
END_ACTION

ACTION A_WaitAtPoint:
stError.POUState := nStateAction;

IF fbComplexAction.bError THEN
	stError.ErrorId :=fbComplexAction.nErrorId;
	nStateAction := 99;
END_IF

CASE nStateAction OF
	0:	//Aktuelles Tool ausgewählt?
		IF stGCodeRef.pCurrentTool = 0 THEN
			stError.Cmd := E_Action.ACTION_MoveToTarget;
			stError.ErrorId := E_ErrorIdGCode.ERRORID_NoSelectedTool;
			nStateAction := 99;
		ELSE
			IF NOT fbItpReadRParams.bBusy THEN
				IF GCode.stGCodeRef.pWaitPoint = 0 THEN
					nStateAction := 2;
				ELSE
					//NCI-Gruppe auflösen
					fbClearGroup(stGCodeRef:= stGCodeRef, bReGearInSlave:= TRUE, bExecute:= TRUE);
					IF NOT fbClearGroup.bBusy THEN
						IF fbClearGroup.bError THEN
							nStateAction := 99;
							stError.ErrorId := fbClearGroup.nErrorId;
						ELSE
							stCurrentPos := pNewTool^.P_stCurrentPosTotal;
							IF bStop THEN
								nStateAction := 80;
							ELSE
								nStateAction := 1;	
							END_IF
						END_IF
						fbClearGroup(stGCodeRef:= stGCodeRef, bExecute:= FALSE);			
					END_IF
				END_IF
			END_IF
		END_IF

	1:	//Action "MoveToTarget" ausführen
		IF bStop THEN
			nStateAction := 80;
			RETURN;
		END_IF	
		MEMSET(ADR(stActionData),0,SIZEOF(stActionData));
		stActionData.eAction := E_Action.ACTION_MoveToTarget;
		stActionData.nObject := stGCodeRef.pCurrentTool^.P_nObjectID;
		stActionData.nTarget := GCode.stGCodeRef.pWaitPoint^.P_nObjectID;
		stActionData.aParams[1] := E_TargetRef.TARGETREF_Center;
		stActionData.aParams[5] := -1;	//SpeedX
		stActionData.aParams[6] := -1;	//SpeedY
		stActionData.aParams[7] := -1; 	//SpeedZ

		stError.ErrorId := fbComplexAction.M_ExeAction(stActionData);
		IF stError.ErrorId > 0 THEN
			nStateAction := 99;
		ELSE
			nStateAction := 2;	
		END_IF
		
	2:	//MoveToTarget ready? -> Warten
		IF bStop THEN
			IF fbComplexAction.bBusy THEN
				fbComplexAction.M_Stop();
			ELSE
				nStateAction := 80;
			END_IF		
		ELSE
			IF NOT fbComplexAction.bBusy THEN
				timer(IN:=TRUE, PT:= LREAL_TO_TIME(alrRParam[1]));
				nStateAction := 3;
			END_IF
		END_IF

	3:	//Warten
		IF bStop THEN
			timer(IN:= FALSE);
			nStateAction := 80;
		ELSE
			timer();
			IF timer.Q THEN
				timer(IN:= FALSE);
				IF GCode.stGCodeRef.pWaitPoint = 0 THEN
					nStateAction := 80;
				ELSE
					nStateAction := 4;	
				END_IF
				
			END_IF
		END_IF
		
	4:	//MoveFree
		A_MoveFree();
		IF nStateA_MoveFree >= 80 THEN
			IF nStateA_MoveFree = 99 THEN
				nStateAction := 99;
			ELSE
				nStateAction := 80;
			END_IF
			nStateA_MoveFree := 0;
		END_IF
END_CASE
END_ACTION

ACTION A_WaitForUser:
stError.POUState := nStateAction;
CASE nStateAction OF
	0:	//R-Parameter einlesen
		IF bStop THEN
			nStateAction := 80;
		ELSE
			IF stGCodeRef.pCurrentTool = 0 THEN
				stError.ErrorId := E_ErrorIdGCode.ERRORID_NoSelectedTool;
				nStateAction := 99;
			ELSE
				IF NOT fbItpReadRParams.bBusy THEN
					//Request absenden
					MEMSET(ADR(stInterResponse),0,SIZEOF(stInterResponse));
					stInteractRequest.eInteractMessageType := E_InteractMessageType.INTERACTMES_WaitForUser;
					stInteractRequest.nObjectId := stGCodeRef.pCurrentTool^.P_nObjectID;
					stInteractRequest.nArg1 := LREAL_TO_DINT(alrRParam[1]);
					stInteractRequest.nArg2 := LREAL_TO_DINT(alrRParam[2]);
					stInteractRequest.nArg3 := LREAL_TO_DINT(alrRParam[3]);
					stInteractRequest.nArg4 := LREAL_TO_DINT(alrRParam[4]);
					nStateAction := 1;
				ELSE
					MEMSET(ADR(stInteractRequest),0,SIZEOF(stInteractRequest));
				END_IF
			END_IF
		END_IF
		
	1:	//auf User Response warten
		IF stInterResponse.eInteractMessageType = E_InteractMessageType.INTERACTMES_Continue OR bStop THEN
			MEMSET(ADR(stInteractRequest),0,SIZEOF(stInteractRequest));
			nStateAction := 80;
		END_IF
END_CASE
END_ACTION

METHOD M_Reset
VAR_INPUT
END_VAR
fbItpReadRParams(sNciToPlc:= stGCodeRef.sNciToPlc, bExecute:= FALSE);
fbItpConfirmHsk(bExecute:= FALSE ,sNciToPlc:= stGCodeRef.sNciToPlc, sPlcToNci:= stGCodeRef.sPlcToNci);
bMFuncRequest := FALSE;
bMFuncConfirm := FALSE;
nStateAction := 0;
bBusy := FALSE;
bCanceled := FALSE;
bError := FALSE;
bStop := FALSE;
timer(IN:= FALSE);
END_METHOD

METHOD M_ValidateTargetNr : BOOL
VAR_INPUT
	nTargetNr 	: UINT;
END_VAR

VAR
	pTarget 	: POINTER TO FB_TargetBase;
END_VAR
IF nTargetNr > 0 AND nTargetNr < GCode.cMaxGCodeTargets THEN
	IF fbObjectDirectory.M_ObjIsTarget(stGCodeRef.aTargetTable[nTargetNr]) THEN
		M_ValidateTargetNr := TRUE;
	END_IF
END_IF
END_METHOD

END_FUNCTION_BLOCK

// ---- Objects/Tools/FB_TwinExtruder.TcPOU
FUNCTION_BLOCK FB_TwinExtruder EXTENDS FB_GCodeTool IMPLEMENTS I_Dispenser
VAR
	pFbHeaterRef	: POINTER TO FB_MZHeaterRef;
	pFirstExtruder 	: POINTER TO FB_Extruder;
	pSecondExtruder	: POINTER TO FB_Extruder;
	///****************************************Aktionvariablen****************************************************
	
	//Action: "Extrude"
	bExtrude			: BOOL;
	nStateA_Extrude		: USINT;
	nExtrudeDistance	: DINT;
	nExtrudeCtrl		: DINT;
	
	nCurrentTemp		: UINT;
END_VAR
VAR CONSTANT
	cNumberOfSlots: UINT := 4; //Slot für Exposure hinzugefügt
END_VAR

SUPER^();	//FB_MzTool aufrufen

IF bExtrude THEN	//Extrudieren
	A_Extrude();
	IF nStateA_Extrude >= 80 THEN
		IF nStateA_Extrude >= 99 THEN
			bError := TRUE;
		END_IF
		bExtrude := FALSE;
		nStateA_Extrude := 0;
		M_RemoveListEntry(nSearchValue:= E_Action.ACTION_Extrude);
	END_IF
END_IF

//Prozessdaten aktualisieren
IF pFbHeaterRef > 0 THEN
	stProcessData.n32Data[7] := BOOL_TO_DINT(pFbHeaterRef^.bHeaterIsOn);
	nCurrentTemp := pFbHeaterRef^.nTemp3Actual;
	stProcessData.n32Data[8] := nCurrentTemp;
END_IF

IF pFirstExtruder > 0 AND pSecondExtruder > 0 THEN
	stProcessData.n32Data[9] := BOOL_TO_DINT(pFirstExtruder^.P_bIsExtruding OR pSecondExtruder^.P_bIsExtruding);
END_IF

aObjProcData[nNotifyId] := stProcessData;

ACTION A_Extrude:
IF pFirstExtruder^.P_bError THEN
	stError.ErrorId := pFirstExtruder^.P_nErrorId;
	stError.POUState := nStateA_Extrude;
	nStateA_Extrude := 99;
END_IF

IF nStateA_Extrude <> 99 THEN
	IF pSecondExtruder^.P_bError THEN
		stError.ErrorId := pSecondExtruder^.P_nErrorId;
		stError.POUState := nStateA_Extrude;
		nStateA_Extrude := 99;
	END_IF	
END_IF

CASE nStateA_Extrude OF
	0:	MEMSET(ADR(stActionData),0,SIZEOF(stActionData));
		stActionData.eAction := E_Action.ACTION_Extrude;
		stActionData.aParams[1] := nExtrudeDistance; 
		stActionData.aParams[2] := nExtrudeCtrl;
		stError.ErrorId := pFirstExtruder^.M_ExeAction(stActionData);
		IF stError.ErrorId = 0 THEN
			stError.ErrorId := pSecondExtruder^.M_ExeAction(stActionData);
			IF stError.ErrorId = 0 THEN
				nStateA_Extrude := 1;
			ELSE //FirstExtruder wieder stoppen
				nStateA_Extrude := 99;
			END_IF
		ELSE
			nStateA_Extrude := 99;
		END_IF
		
	1:	//ready ?
		IF NOT(pFirstExtruder^.M_GetActionBusy(E_Action.ACTION_Extrude) OR 
				pSecondExtruder^.M_GetActionBusy(E_Action.ACTION_Extrude)) THEN
			nStateA_Extrude := 80;
		END_IF
		
	70:	//Stoppen
		pFirstExtruder^.M_CancelAction(E_Action.ACTION_Extrude);
		pSecondExtruder^.M_CancelAction(E_Action.ACTION_Extrude);
		nStateA_Extrude := 71;
		
	71:	IF NOT(pFirstExtruder^.M_GetActionBusy(E_Action.ACTION_Extrude) OR 
			pSecondExtruder^.M_GetActionBusy(E_Action.ACTION_Extrude)) THEN
			nStateA_Extrude := 80;
		END_IF
END_CASE

IF nStateA_Extrude = 99 THEN
	pFirstExtruder^.M_CancelAction(E_Action.ACTION_Extrude);
	pSecondExtruder^.M_CancelAction(E_Action.ACTION_Extrude);
	stError.Cmd := E_Action.ACTION_Extrude;
	stError.POU := E_POU.POU_FB_TwinExtruder;
	stError.POUAction := E_POUACT.POUACT_A_Extrude;
	fbErrorList.M_Add(stError);	
END_IF
END_ACTION

ACTION A_Reset:
nStateA_ResetSpec := 80;
SUPER^.A_Reset();
END_ACTION

ACTION A_Stop:
IF nStateA_Stop = 0 THEN

	nStateA_Stop := 1;
END_IF

SUPER^.A_Stop();
END_ACTION

METHOD FB_init : BOOL
VAR_INPUT
	bInitRetains : BOOL; // if TRUE, the retain variables are initialized (warm start / cold start)
	bInCopyCode : BOOL;  // if TRUE, the instance afterwards gets moved into the copy code (online change)
END_VAR
eObjectType := E_ObjectType.OBJECTTYPE_TwinExtruder;
eObjectGroup := E_ObjectGroup.OBJECTGROUP_MzTool OR E_ObjectGroup.OBJECTGROUP_Device;
END_METHOD

METHOD M_AddChild : ERRORID
VAR_INPUT
	pObject : POINTER TO FB_Object;
	nSlotNr	: UINT;
	nIndex 	: INT;
END_VAR
//Kann folgende Objekt-Typen aufnehmen
//Extruder, Nozzle, Exposure
IF pObject > 0 THEN
	IF pObject^.P_eObjectType = E_ObjectType.OBJECTTYPE_Extruder OR
		pObject^.P_eObjectType = E_ObjectType.OBJECTTYPE_DummyTool OR
		pObject^.P_eObjectType = E_ObjectType.OBJECTTYPE_Exposure OR
		pObject^.P_eObjectType = E_ObjectType.OBJECTTYPE_Nozzle THEN
		M_AddChild := SUPER^.M_AddChild(pObject,nSlotNr,nIndex);
	ELSE
		M_AddChild := E_ErrorIdObjMgmt.ERRORID_InvalidParentObject;
	END_IF
ELSE
	M_AddChild := E_ErrorIdObjMgmt.ERRORID_InvalidParentObject;
END_IF
END_METHOD

METHOD M_CancelAction
VAR_INPUT
	eAction : E_Action;
END_VAR
IF eAction = E_Action.ACTION_Extrude THEN
	IF bExtrude AND nStateA_Extrude < 70 THEN
		nStateA_Extrude := 70;
	END_IF
ELSE
	SUPER^.M_CancelAction(eAction);
END_IF
END_METHOD

METHOD M_CheckAction : ERRORID
VAR_INPUT
	refActionData	: REFERENCE TO ST_ActionData;
	pCorrelObject	: POINTER TO FB_Object;
END_VAR
CASE refActionData.eAction OF
	E_Action.ACTION_Extrude, //BasicAction für ActionOnArray
	E_Action.ACTION_CleanTip,
	E_Action.ACTION_MeasureTool,
	E_Action.ACTION_TeachTarget:
		RETURN;
ELSE
	M_CheckAction := SUPER^.M_CheckAction(refActionData, pCorrelObject);
END_CASE
END_METHOD

METHOD M_CheckProcDataType : BOOL
VAR_INPUT
	eProcDataType : E_ProcDataType;
END_VAR
IF eProcDataType = E_ProcDataType.PROCDATATYPE_Temp1 THEN
	M_CheckProcDataType := TRUE;
END_IF
END_METHOD

METHOD M_CheckProps : ERRORID
VAR_INPUT
END_VAR

VAR
	pSlot : POINTER TO FB_Slot;
END_VAR
M_CheckProps := SUPER^.M_CheckProps();
//TwinExtruder muss zwingend zwei Childs als Extruder besitzen
//auf Slot1 -> FirstExtruder
//auf Slot2 -> SecondExtruder
pFirstExtruder := 0;
pSecondExtruder := 0;

pSlot := fbSlotList.M_GetAtNr(1);
IF pSlot > 0 THEN
	IF pSlot^.P_pChild > 0 THEN
		IF pSlot^.P_pChild^.P_eObjectType = E_ObjectType.OBJECTTYPE_Extruder THEN
			pFirstExtruder := pSlot^.P_pChild;
		END_IF
	END_IF
END_IF

pSlot := fbSlotList.M_GetAtNr(2);
IF pSlot > 0 THEN
	IF pSlot^.P_pChild > 0 THEN
		IF pSlot^.P_pChild^.P_eObjectType = E_ObjectType.OBJECTTYPE_Extruder THEN
			pSecondExtruder := pSlot^.P_pChild;
		END_IF
	END_IF
END_IF

IF pFirstExtruder = 0 OR pSecondExtruder = 0 THEN
	M_CheckProps := E_ErrorIdObjMgmt.ERRORID_UnusedExtruderSlot;
END_IF

IF pPiece = 0 THEN
	M_CheckProps := E_ErrorIdObjMgmt.ERRORID_NoNozzleOnTool;
END_IF
END_METHOD

METHOD M_DispenserPrepare : ERRORID
VAR_INPUT
END_VAR
END_METHOD

METHOD M_DispenserStart : ERRORID
VAR_INPUT
END_VAR

VAR
	stActionData : ST_ActionData;
END_VAR
stActionData.eAction := E_ACTION.ACTION_Extrude;
stActionData.aParams[2] := 1;
M_DispenserStart := M_ExeAction(stActionData);
END_METHOD

METHOD M_DispenserStop : ERRORID
VAR_INPUT
END_VAR

VAR
	stActionData : ST_ActionData;
END_VAR
stActionData.eAction := E_ACTION.ACTION_Extrude;
M_DispenserStop := M_ExeAction(stActionData);
END_METHOD

METHOD M_ExeAction : ERRORID
VAR_INPUT
	refActionData : REFERENCE TO ST_ActionData;	
END_VAR
IF NOT (eCurrentState = E_MachineState.MACHINESTATE_Idle OR
	eCurrentState = E_MachineState.MACHINESTATE_Active OR
	eCurrentState = E_MachineState.MACHINESTATE_Ready) THEN
	M_ExeAction := E_ErrorIdCmd.ERRORID_InvalidState;
	RETURN;
END_IF

CASE refActionData.eAction OF
		E_Action.ACTION_Extrude:
			//Beide Extruder gelockt?
			IF NOT (pFirstExtruder^.P_bIsLocked AND pSecondExtruder^.P_bIsLocked) THEN
				M_ExeAction := E_ErrorIdCmd.ERRORID_DeviceNotLocked;
				RETURN;				
			END_IF
			
			nExtrudeDistance := refActionData.aParams[1]; 
			nExtrudeCtrl := refActionData.aParams[2];
			
			IF NOT bExtrude AND nExtrudeCtrl = 1 THEN //Einschalten
				bExtrude := TRUE;
				fbList.A_AddHeadValue(hList := hList, putValue := E_Action.ACTION_Extrude);
			ELSIF bExtrude AND nExtrudeCtrl = 0 THEN //Ausschalten
				MEMSET(ADR(stActionData),0,SIZEOF(stActionData));
				stActionData.eAction := E_Action.ACTION_Extrude;
				stActionData.aParams[1] := nExtrudeDistance; 
				stActionData.aParams[2] := nExtrudeCtrl := 0; 
				pFirstExtruder^.M_ExeAction(stActionData);
				pSecondExtruder^.M_ExeAction(stActionData);
			ELSE
				RETURN;
			END_IF
			
	ELSE
		M_ExeAction := SUPER^.M_ExeAction(refActionData);
		RETURN;
END_CASE

bBusy := TRUE;
eCurrentState := E_MachineState.MACHINESTATE_Active;
END_METHOD

METHOD M_GetAllProps : ERRORID
VAR_INPUT
	refCmdData : REFERENCE TO  ST_CmdData;
END_VAR

VAR
	i : UINT;
	pToolSlot	: POINTER TO FB_Slot;
END_VAR
//BaseProperties lesen
SUPER^.M_GetAllProps(refCmdData);

nCurrentPropIndex := nCurrentPropIndex + 1;
IF pFbHeaterRef > 0 THEN
	refCmdData.n32Data[nCurrentPropIndex] := 1;	
END_IF
END_METHOD

METHOD M_GetProcData : DINT
VAR_INPUT
	eProcDataType : E_ProcDataType;
END_VAR
IF eProcDataType = E_ProcDataType.PROCDATATYPE_Temp1 THEN
	M_GetProcData := nCurrentTemp;
END_IF
END_METHOD

METHOD M_SetAllProps : ERRORID
VAR_INPUT
	refCmdData : REFERENCE TO  ST_CmdData;
END_VAR

VAR
	nParentMzToolObjId	: UINT;
	pParentTool 		: POINTER TO FB_MzTool;
	pParentHead 		: POINTER TO FB_MzHead;
END_VAR
M_SetAllProps := SUPER^.M_SetAllProps(refCmdData);

IF M_SetAllProps > 0 THEN
	RETURN;
END_IF

//Spezi-Paramter schreiben
nCurrentPropIndex := nCurrentPropIndex + 1;
nSpecPropIndex := nCurrentPropIndex;

IF refCmdData.n32Data[nCurrentPropIndex] = 1 THEN
	pFbHeaterRef := ADR(pFbMultiZ^.aFbHeaterRef[7]);
ELSE
	pFbHeaterRef := 0;
END_IF

nNoOfProps := nCurrentPropIndex + 1;
END_METHOD

METHOD M_SetPrintParams : ST_MethResult
VAR_INPUT
	eType 		: E_PrintParamType;
	nNumerator	: USINT;
	nValue		: DINT;
END_VAR

VAR
	stActionData : ST_ActionData;
END_VAR
IF eType = E_PrintParamType.Feed THEN
	IF nNumerator = 1 THEN
		IF pFirstExtruder > 0 THEN
			M_SetPrintParams.nErrorId := pFirstExtruder^.M_SetFeed(DINT_TO_UINT(nValue));	
		END_IF	
	ELSIF nNumerator = 2 THEN
		IF pSecondExtruder > 0 THEN
			M_SetPrintParams.nErrorId := pSecondExtruder^.M_SetFeed(DINT_TO_UINT(nValue));	
		END_IF	
	ELSE
		M_SetPrintParams.nErrorId := E_ErrorIdCmd.ERRORID_InvalidPrintParamNumerator;
	END_IF
ELSE
	M_SetPrintParams.nErrorId := E_ErrorIdCmd.ERRORID_InvalidPrintParamType;
END_IF

IF M_SetPrintParams.nErrorId > 0 THEN
	M_SetPrintParams.bError := TRUE;
END_IF
END_METHOD

PROPERTY P_bSensorMounted : BOOL
GET
P_bSensorMounted:= pFirstExtruder^.P_bSensorMounted OR pSecondExtruder^.P_bSensorMounted;
END_GET
END_PROPERTY

PROPERTY P_eDispenserState : E_DispenserState
GET
IF pFirstExtruder > 0 AND_THEN pFirstExtruder^.P_bIsExtruding THEN
	P_eDispenserState := E_DispenserState.Dispensing;
END_IF

IF pSecondExtruder > 0 AND_THEN pSecondExtruder^.P_bIsExtruding THEN
	P_eDispenserState := E_DispenserState.Dispensing;
END_IF
END_GET
END_PROPERTY

PROPERTY P_pFirstExtruder : POINTER TO FB_Extruder
GET
P_pFirstExtruder := pFirstExtruder;
END_GET
END_PROPERTY

PROPERTY P_pSecondExtruder : POINTER TO FB_Extruder
GET
P_pSecondExtruder := pSecondExtruder;
END_GET
END_PROPERTY

END_FUNCTION_BLOCK

// ---- Objects/Tools/FB_MultiCartHolder.TcPOU
FUNCTION_BLOCK FB_MultiCartHolder EXTENDS FB_GCodeTool IMPLEMENTS I_Dispenser
VAR_INPUT
END_VAR
VAR_OUTPUT
END_VAR
VAR
	//Specproperties
	pFbHeaterRef		: POINTER TO FB_MZHeaterRef;
	pCartDispenser1		: POINTER TO FB_CartDispenser;
	pCartDispenser2		: POINTER TO FB_CartDispenser;
	pCartDispenser3		: POINTER TO FB_CartDispenser;

	//****************************************Aktionsvariablen****************************************************

	//Action: "SwitchPressure"
	//Diese Action wird auf alle vorhandene Childs vom Typ CartridgeDispenser ausgeführt
	//es werden also Zeiger auf die entpsrechende Tools gesetzt
	//Die Frage ist, wie man das mit der Zeit macht? Na genauso wie bei den einzelnen.
	bSwitchPress		: BOOL;			
	nStateA_SwitchPress	: USINT;		//State von A_SwitchPress()
	eSwitchPressCtrl	: E_PressCtrl;
	tPressTime			: TIME;			//nach dieser Zeit Ventil automatisch wieder zu
	timerPress			: TON;			//Timer für Öffnungszeit Druckventil
	bPressIsOn			: BOOL;	
	
	
	
	//Action: "Heating"
	bHeating 			: BOOL;
	nStateA_Heating		: USINT;		//State von A_Heating()
	nTempSetpoint		: UINT;			//Solltemperatur
	bHeatingOn			: BOOL;			//Heizung "EIN"
	fbHeaterCtrl		: FB_MzHeaterControl;
	
	nCurrentTemp1		: UINT;
	nCurrentTemp2		: UINT;
END_VAR

VAR CONSTANT
	cHotTemp		: UINT := 500;	//ab dieser Isttemperatur wird Tool als heiß betrachtet (Interlock)
END_VAR

IF eCurrentState = E_MachineState.MACHINESTATE_Active THEN
	IF bHeating THEN	//Heizen
		A_Heating();
		IF nStateA_Heating >= 80 THEN
			IF nStateA_Heating >= 99 THEN
				bError := TRUE;
			END_IF
			M_RemoveListEntry(nSearchValue:= E_Action.ACTION_Heating);
			bHeating := FALSE;
			nStateA_Heating := 0;
		END_IF
	END_IF
	
	IF bSwitchPress THEN	//Kartuschendruck einstellen und Ein-bzw. Aus schalten 
		A_SwitchPress();
		IF nStateA_SwitchPress >= 80 THEN
			IF nStateA_SwitchPress >= 99 THEN
				bError := TRUE;
			END_IF
			bSwitchPress := FALSE;
			nStateA_SwitchPress := 0;
			M_RemoveListEntry(nSearchValue:= E_Action.ACTION_SwitchPressure);
		END_IF
	END_IF

	
END_IF

SUPER^();	//FB_MzTool aufrufen

//Prozessdaten aktualisieren
IF pZAxisRef > 0 THEN
	stProcessData.n32Data[7] := BOOL_TO_DINT(pZAxisRef^.stInput.nToolState.2);
	//Komplett überarbeiten
END_IF

aObjProcData[nNotifyId] := stProcessData;

ACTION A_Heating:
IF nStateA_Heating = 0 THEN
	fbHeaterCtrl(bExecute:= TRUE, nTempZone1:= nTempSetpoint, bHeatingOn:= bHeatingOn, pFbHeaterRef:= pFbHeaterRef);

	IF NOT fbHeaterCtrl.bBusy THEN
		IF fbHeaterCtrl.bError THEN
			stError.ErrorId := fbHeaterCtrl.nErrorId; 
			stError.POUState := nStateA_Heating;
			nStateA_Heating := 99;
		ELSE
			nStateA_Heating := 80;	
		END_IF
		fbHeaterCtrl(bExecute:= FALSE, pFbHeaterRef:= pFbHeaterRef);
	END_IF
ELSIF nStateA_Heating = 70 THEN
	fbHeaterCtrl(bExecute:= FALSE, pFbHeaterRef:= pFbHeaterRef);
	nStateA_Heating := 80;
END_IF

//Errorhandling
IF nStateA_Heating = 99 THEN
	stError.POU := E_POU.POU_FB_MultiCartHolder;
	stError.Cmd := E_Action.ACTION_Heating;
	stError.POUAction := E_POUACT.POUACT_A_Heating;
	fbErrorList.M_Add(stError);
END_IF
END_ACTION

ACTION A_Reset:
//Ist noch eine Aktion aktiv?
IF nStateA_ResetSpec = 0 THEN 
	IF bHeating THEN
		bHeating := FALSE;
		nStateA_Heating := 0;
	END_IF
	
	nStateA_ResetSpec := 80;
END_IF

SUPER^.A_Reset();
END_ACTION

ACTION A_Stop:
IF nStateA_Stop = 0 THEN
	nStateA_Stop := 1;	
END_IF

SUPER^.A_Stop();
END_ACTION

ACTION A_SwitchPress:
CASE nStateA_SwitchPress OF
	0: 
		IF pCartDispenser1 > 0 THEN
			IF pCartDispenser1^.M_GetActionBusy(E_Action.ACTION_SwitchPressure) THEN
				RETURN;
			END_IF
		END_IF
		IF pCartDispenser2 > 0 THEN
			IF pCartDispenser2^.M_GetActionBusy(E_Action.ACTION_SwitchPressure) THEN
				RETURN;
			END_IF
		END_IF
		IF pCartDispenser3 > 0 THEN
			IF pCartDispenser3^.M_GetActionBusy(E_Action.ACTION_SwitchPressure) THEN
				RETURN;
			END_IF
		END_IF
		nStateA_SwitchPress := 80;
	
	70:
		IF pCartDispenser1 > 0 THEN
			pCartDispenser1^.M_CancelAction(E_Action.ACTION_SwitchPressure);
		END_IF
		IF pCartDispenser2 > 0 THEN
			pCartDispenser2^.M_CancelAction(E_Action.ACTION_SwitchPressure);
		END_IF
		IF pCartDispenser3 > 0 THEN
			pCartDispenser3^.M_CancelAction(E_Action.ACTION_SwitchPressure);
		END_IF
		nStateA_SwitchPress := 80;
END_CASE
END_ACTION

METHOD FB_init : BOOL
VAR_INPUT
	bInitRetains : BOOL; // if TRUE, the retain variables are initialized (warm start / cold start)
	bInCopyCode : BOOL;  // if TRUE, the instance afterwards gets moved into the copy code (online change)
END_VAR
eObjectType := E_ObjectType.OBJECTTYPE_MultiCartHolder;
eObjectGroup := E_ObjectGroup.OBJECTGROUP_MzTool OR E_ObjectGroup.OBJECTGROUP_Device;
END_METHOD

METHOD M_AddChild : ERRORID
VAR_INPUT
	pObject : POINTER TO FB_Object;
	nSlotNr	: UINT;
	nIndex : INT;
END_VAR
IF pObject > 0 THEN
	IF pObject^.P_eObjectType = E_ObjectType.OBJECTTYPE_CartDispenser OR
		pObject^.P_eObjectType = E_ObjectType.OBJECTTYPE_CartDispStirrer OR
		pObject^.P_eObjectType = E_ObjectType.OBJECTTYPE_DummyTool OR
		pObject^.P_eObjectType = E_ObjectType.OBJECTTYPE_Nozzle THEN
		M_AddChild := SUPER^.M_AddChild(pObject,nSlotNr,nIndex);
	ELSE
		M_AddChild := E_ErrorIdObjMgmt.ERRORID_InvalidParentObject;
	END_IF
ELSE
	M_AddChild := E_ErrorIdObjMgmt.ERRORID_InvalidParentObject;
END_IF
END_METHOD

METHOD M_CancelAction
VAR_INPUT
	eAction : E_Action;
END_VAR
CASE eAction OF
	E_Action.ACTION_Heating:
		IF bHeating AND nStateA_Heating < 70 THEN
			nStateA_Heating := 70;
		END_IF

	E_Action.ACTION_SwitchPressure:
		//es stellt sich die Frage, ob das notwendig ist, da ja eventuell bei den Childs abgebrochen wird

ELSE
	SUPER^.M_CancelAction(eAction);
END_CASE
END_METHOD

METHOD M_CheckAction : ERRORID
VAR_INPUT
	refActionData 	: REFERENCE TO ST_ActionData;
	pCorrelObject	: POINTER TO FB_Object;
END_VAR
CASE refActionData.eAction OF
	E_Action.ACTION_CleanTip,
	E_Action.ACTION_MeasureTool,
	E_Action.ACTION_SwitchPressure, //BasicAction für ActionOnArray
	E_Action.ACTION_TeachTarget:
		RETURN;
ELSE
	M_CheckAction := SUPER^.M_CheckAction(refActionData, pCorrelObject);
END_CASE
END_METHOD

METHOD M_CheckProcDataType : BOOL
VAR_INPUT
	eProcDataType : E_ProcDataType;
END_VAR
IF eProcDataType = E_ProcDataType.PROCDATATYPE_Temp1 OR eProcDataType = E_ProcDataType.PROCDATATYPE_Temp2 THEN
	M_CheckProcDataType := TRUE;
END_IF
END_METHOD

METHOD M_CheckProps : ERRORID
VAR_INPUT
END_VAR

VAR
	i : UINT;
	pSlot : POINTER TO FB_Slot;
END_VAR
M_CheckProps := SUPER^.M_CheckProps();
//Kann bis zu 3 CartDispenser enthalten
pCartDispenser1 := 0;
pCartDispenser2	:= 0;
pCartDispenser3	:= 0;
FOR i:= 1 TO nNumberOfSlots BY 1 DO
	pSlot := fbSlotList.M_GetAtNr(i);
	IF pSlot > 0 AND_THEN pSlot^.P_pChild > 0 AND_THEN
		(pSlot^.P_pChild^.P_eObjectType = E_ObjectType.OBJECTTYPE_CartDispenser OR pSlot^.P_pChild^.P_eObjectType = E_ObjectType.OBJECTTYPE_CartDispStirrer) THEN
		CASE pSlot^.P_nNr OF
			1: pCartDispenser1 := pSlot^.P_pChild;
			2: pCartDispenser2 := pSlot^.P_pChild;
			3: pCartDispenser3 := pSlot^.P_pChild;
		END_CASE
	END_IF
END_FOR

IF pPiece = 0 THEN
	M_CheckProps := E_ErrorIdObjMgmt.ERRORID_NoNozzleOnTool;
END_IF
END_METHOD

METHOD M_ClearAllProps
VAR_INPUT
	bIgnoreParent : BOOL; //Es wird das gesamte OD gelöscht. -> Zeiger auf Parent nicht mehr gültig!
END_VAR
pCartDispenser1 := 0;
pCartDispenser2 := 0;
pCartDispenser3 := 0;
SUPER^.M_ClearAllProps(bIgnoreParent);
END_METHOD

METHOD M_DispenserPrepare : ERRORID
VAR_INPUT
END_VAR
END_METHOD

METHOD M_DispenserStart : ERRORID
VAR_INPUT
END_VAR

VAR
	stActionData : ST_ActionData;
END_VAR
//Es werden alle 3 Kartuschen (wenn vorhanden) dauerhaft eingeschalten
stActionData.eAction := E_Action.ACTION_SwitchPressure;
stActionData.aParams[1] := 7;
M_DispenserStart := M_ExeAction(stActionData);
END_METHOD

METHOD M_DispenserStop : ERRORID
VAR_INPUT
END_VAR

VAR
	stActionData : ST_ActionData;
END_VAR
stActionData.eAction := E_Action.ACTION_SwitchPressure;
M_DispenserStop := M_ExeAction(stActionData);
END_METHOD

METHOD M_ExeAction : ERRORID
VAR_INPUT
	refActionData : REFERENCE TO ST_ActionData;	
END_VAR

VAR
	bFlag : BOOL;
	stActionData : ST_ActionData;
	tPressTime : TIME;
END_VAR
IF NOT (eCurrentState = E_MachineState.MACHINESTATE_Idle OR
	eCurrentState = E_MachineState.MACHINESTATE_Active OR
	eCurrentState = E_MachineState.MACHINESTATE_Ready) THEN
	M_ExeAction := E_ErrorIdCmd.ERRORID_InvalidState;
	RETURN;
END_IF

CASE refActionData.eAction OF
	E_Action.ACTION_Heating:
		IF nStateA_Heating = 0 THEN
			nTempSetpoint := DINT_TO_UINT(refActionData.aParams[1]);
			IF nTempSetpoint > 2000 THEN
				M_ExeAction := E_ErrorIdCmd.ERRORID_InvalidHeatingTemp;  //Error
				RETURN;
			END_IF
			bHeatingOn := DINT_TO_BOOL(refActionData.aParams[2]);			
			bHeating := TRUE;
			fbList.A_AddHeadValue(hList := hList, putValue := E_Action.ACTION_Heating);
		ELSE
			RETURN;
		END_IF
		
	E_Action.ACTION_SwitchPressure:
		//Die Action kann nur ausgeführt werden, wenn es mind. ein Child vom Typ "CartDispenser" gibt.
		//Die einzelnen Bits aus aParams[1] werden als die einzelnen Dispenser angesehen
		IF pCartDispenser1 > 0 OR pCartDispenser2 > 0 OR pCartDispenser3 > 0 THEN
			//Die einzelnen Bits extrahieren
			tPressTime := DINT_TO_TIME(refActionData.aParams[2]);
			IF pCartDispenser1 > 0 THEN
				IF refActionData.aParams[1].0 THEN
					M_ExeAction := pCartDispenser1^.M_SwitchPressure(E_PressCtrl.PRESSCTRL_PressOn,tPressTime);
				ELSE
					M_ExeAction := pCartDispenser1^.M_SwitchPressure(E_PressCtrl.PRESSCTRL_Off,tPressTime);
				END_IF
				IF M_ExeAction > 0 THEN
					RETURN;
				END_IF
				IF pCartDispenser1^.M_GetActionBusy(E_Action.ACTION_SwitchPressure) THEN
					bFlag := TRUE;
				END_IF				
			END_IF
			
			IF pCartDispenser2 > 0 THEN
				IF refActionData.aParams[1].1 THEN
					M_ExeAction := pCartDispenser2^.M_SwitchPressure(E_PressCtrl.PRESSCTRL_PressOn,tPressTime);
				ELSE
					M_ExeAction := pCartDispenser2^.M_SwitchPressure(E_PressCtrl.PRESSCTRL_Off,tPressTime);
				END_IF
				IF M_ExeAction > 0 THEN
					RETURN;
				END_IF
				IF pCartDispenser2^.M_GetActionBusy(E_Action.ACTION_SwitchPressure) THEN
					bFlag := TRUE;
				END_IF				
			END_IF
			
			IF pCartDispenser3 > 0 THEN
				IF refActionData.aParams[1].2 THEN
					M_ExeAction := pCartDispenser3^.M_SwitchPressure(E_PressCtrl.PRESSCTRL_PressOn,tPressTime);
				ELSE
					M_ExeAction := pCartDispenser3^.M_SwitchPressure(E_PressCtrl.PRESSCTRL_Off,tPressTime);
				END_IF
				IF M_ExeAction > 0 THEN
					RETURN;
				END_IF
				IF pCartDispenser3^.M_GetActionBusy(E_Action.ACTION_SwitchPressure) THEN
					bFlag := TRUE;
				END_IF				
			END_IF
			
			IF bFlag AND NOT bSwitchPress THEN
				bSwitchPress := TRUE;
				fbList.A_AddHeadValue(hList := hList, putValue := E_Action.ACTION_SwitchPressure);
			END_IF
		
		ELSE
			M_ExeAction := E_ErrorIdCmd.ERRORID_NoCartridgeDispConfigured;
			RETURN;			
		END_IF

	ELSE
		M_ExeAction := SUPER^.M_ExeAction(refActionData);
		RETURN;
END_CASE

bBusy := TRUE;
eCurrentState := E_MachineState.MACHINESTATE_Active;
END_METHOD

METHOD M_GetAllProps : ERRORID
VAR_INPUT
	refCmdData : REFERENCE TO  ST_CmdData;
END_VAR
//Basisproperties lesen
SUPER^.M_GetAllProps(refCmdData);
//Specialproperties lesen
nCurrentPropIndex := nCurrentPropIndex + 1;
refCmdData.n32Data[nCurrentPropIndex] := BOOL_TO_DINT(pFbHeaterRef^.P_bHeaterDetected);
END_METHOD

METHOD M_GetProcData : DINT
VAR_INPUT
	eProcDataType : E_ProcDataType;
END_VAR
IF eProcDataType = E_ProcDataType.PROCDATATYPE_Temp1 THEN
	M_GetProcData := nCurrentTemp1;
ELSIF eProcDataType = E_ProcDataType.PROCDATATYPE_Temp2 THEN
	M_GetProcData := nCurrentTemp2;
END_IF
END_METHOD

METHOD M_SetAllProps : ERRORID
VAR_INPUT
	refCmdData : REFERENCE TO  ST_CmdData;
END_VAR
M_SetAllProps := SUPER^.M_SetAllProps(refCmdData);

IF M_SetAllProps > 0 THEN
	RETURN;
END_IF

nCurrentPropIndex := nCurrentPropIndex + 1;
nSpecPropIndex := nCurrentPropIndex;

pFbHeaterRef := ADR(pFbMultiZ^.aFbHeaterRef[pZAxisRef^.nChannel]);
pFbHeaterRef^.P_bHeaterDetected := DINT_TO_BOOL(refCmdData.n32Data[nCurrentPropIndex]);

IF pFbHeaterRef^.P_bHeaterDetected THEN
	pZAxisRef^.eFixedToolType := E_MzToolType.TOOL_TYPE_Cartridge;
ELSE
	pZAxisRef^.eFixedToolType := E_MzToolType.TOOL_TYPE_None;
END_IF

nNoOfProps := nCurrentPropIndex + 1;
END_METHOD

METHOD M_SetPrintParams : ST_MethResult
VAR_INPUT
	eType 		: E_PrintParamType;
	nNumerator	: USINT;
	nValue		: DINT;
END_VAR

VAR
	stActionData : ST_ActionData;
	pCurrentDispenser : POINTER TO FB_CartDispenser;
END_VAR

VAR_STAT
	bExecuted : BOOL;
END_VAR
stActionData.eAction := E_Action.ACTION_SetPressure;
stActionData.aParams[2] := nValue; //Soll

IF eType = E_PrintParamType.Pressure THEN
	CASE nNumerator OF
		1:	pCurrentDispenser := pCartDispenser1;
		
		2:	pCurrentDispenser := pCartDispenser2;
		
		3:	pCurrentDispenser := pCartDispenser2;
	ELSE
		M_SetPrintParams.bError := TRUE;
		M_SetPrintParams.nErrorId := E_ErrorIdCmd.ERRORID_InvalidPrintParamNumerator;
	END_CASE
ELSE
	M_SetPrintParams.bError := TRUE;
	M_SetPrintParams.nErrorId := E_ErrorIdCmd.ERRORID_InvalidPrintParamType;
	RETURN;		
END_IF

IF pCurrentDispenser = 0 THEN
	M_SetPrintParams.bError := TRUE;
	M_SetPrintParams.nErrorId := E_ErrorIdCmd.ERRORID_InvalidPrintParamNumerator;
	RETURN;
END_IF
  
IF NOT pCurrentDispenser^.P_bPressIsOn THEN
	stActionData.aParams[1] := 1; //Fertigmeldung, wenn Druck erreicht	
	stActionData.aParams[3] := 20; //Toleranz +
	stActionData.aParams[4] := 20; //Toleranz -
	stActionData.aParams[5] := 20000; //Timeout	
END_IF
	
IF NOT bExecuted THEN
	M_SetPrintParams.nErrorId := pCurrentDispenser^.M_ExeAction(stActionData);
	bExecuted := TRUE;
END_IF

IF M_SetPrintParams.nErrorId > 0 THEN
	M_SetPrintParams.bError := TRUE;
ELSIF pCurrentDispenser^.M_GetActionBusy(E_Action.ACTION_SetPressure) THEN //ist ActionStatemachine zur Überwachung gegangen
	M_SetPrintParams.bBusy := TRUE;
	RETURN;
END_IF

bExecuted := FALSE;
END_METHOD

PROPERTY P_bIsHot : BOOL
GET
P_bIsHot := (nCurrentTemp1 >= cHotTemp) OR (nCurrentTemp2 >= cHotTemp);
END_GET
END_PROPERTY

PROPERTY P_eDispenserState : E_DispenserState
GET
IF pCartDispenser1 > 0 AND_THEN pCartDispenser1^.P_bPressIsOn THEN
	P_eDispenserState := E_DispenserState.Dispensing;
END_IF

IF pCartDispenser2 > 0 AND_THEN pCartDispenser2^.P_bPressIsOn THEN
	P_eDispenserState := E_DispenserState.Dispensing;
END_IF

IF pCartDispenser3 > 0 AND_THEN pCartDispenser3^.P_bPressIsOn THEN
	P_eDispenserState := E_DispenserState.Dispensing;
END_IF
END_GET
END_PROPERTY

PROPERTY P_pCartDispenser1 : POINTER TO FB_CartDispenser
GET
P_pCartDispenser1 := pCartDispenser1;
END_GET
END_PROPERTY

PROPERTY P_pCartDispenser2 : POINTER TO FB_CartDispenser
GET
P_pCartDispenser2 := pCartDispenser2;
END_GET
END_PROPERTY

PROPERTY P_pCartDispenser3 : POINTER TO FB_CartDispenser
GET
P_pCartDispenser3 := pCartDispenser3;
END_GET
END_PROPERTY

END_FUNCTION_BLOCK

// ---- Objects/Targets/Passive/FB_VialRack.TcPOU
FUNCTION_BLOCK FB_VialRack EXTENDS FB_Rack
VAR
	nGCodeTargetNr	: UINT;
END_VAR

METHOD FB_init : BOOL
VAR_INPUT
	bInitRetains : BOOL; // if TRUE, the retain variables are initialized (warm start / cold start)
	bInCopyCode : BOOL;  // if TRUE, the instance afterwards gets moved into the copy code (online change)
END_VAR
eObjectType := E_ObjectType.OBJECTTYPE_VialRack;
eObjectGroup := E_ObjectGroup.OBJECTGROUP_Target OR E_ObjectGroup.OBJECTGROUP_Rack;
END_METHOD

METHOD M_AddChild : ERRORID
VAR_INPUT
	pObject : POINTER TO FB_Object;
	nSlotNr	: UINT;
	nIndex 	: INT;
END_VAR
//Kann folgende Objekte aufnehmen:
//Point, Vials
IF pObject > 0 THEN
	IF pObject^.P_eObjectType = E_ObjectType.OBJECTTYPE_Point THEN
		M_AddChild := SUPER^.M_AddChild(pObject,nSlotNr,nIndex);
	ELSIF pObject^.P_eObjectType = E_ObjectType.OBJECTTYPE_Vial OR
			pObject^.P_eObjectType = E_ObjectType.OBJECTTYPE_VialClosed THEN
		//darf nur in ein Slot
		IF nSlotNr > 0 THEN
			M_AddChild := SUPER^.M_AddChild(pObject,nSlotNr,nIndex);
		ELSE
			M_AddChild := E_ErrorIdObjMgmt.ERRORID_InvalidSlotNumber;	
		END_IF
	ELSE
		M_AddChild := E_ErrorIdObjMgmt.ERRORID_InvalidParentObject;
	END_IF
ELSE
	M_AddChild := E_ErrorIdObjMgmt.ERRORID_InvalidParentObject;
END_IF
END_METHOD

METHOD M_CheckAction : ERRORID
VAR_INPUT
	refActionData 	: REFERENCE TO ST_ActionData;
	pCorrelObject	: POINTER TO FB_Object;
END_VAR

VAR
	pSlot : POINTER TO FB_PieceSlot;
	pVial : POINTER TO FB_Vial;
	pMzTool : POINTER TO FB_MzTool;
END_VAR
IF refActionData.eAction = E_Action.ACTION_InsertTool THEN
	pSlot := super^.M_GetSlot(DINT_TO_UINT(refActionData.aParams[2]));
	IF pSlot = 0 THEN
		M_CheckAction := E_ErrorIdCmd.ERRORID_InvalidTargetSlot;
	ELSE
		//Vial in Slot ?
		pVial := pSlot^.P_pPiece;
		IF pVial = 0 THEN
			M_CheckAction := E_ErrorIdCmd.ERRORID_NoPieceInSlot;
		END_IF
	END_IF
ELSIF refActionData.eAction = E_Action.ACTION_DockTool THEN
	pSlot := super^.M_GetSlot(DINT_TO_UINT(refActionData.aParams[2]));
	IF pSlot = 0 THEN
		M_CheckAction := E_ErrorIdCmd.ERRORID_InvalidTargetSlot;
	ELSE
		//Vial in Slot ?
		pVial := pSlot^.P_pPiece;
		IF pVial = 0 THEN
			M_CheckAction := E_ErrorIdCmd.ERRORID_NoPieceInSlot;
		ELSE
			IF pVial^.P_eObjectType = E_ObjectType.OBJECTTYPE_VialClosed THEN
				M_CheckAction := E_ErrorIdCmd.ERRORID_InvalidPieceType;
			END_IF
		END_IF
	END_IF
ELSIF refActionData.eAction = E_Action.ACTION_MeasurepH THEN
	pSlot := super^.M_GetSlot(DINT_TO_UINT(refActionData.aParams[1]));
	IF pSlot = 0 THEN
		M_CheckAction := E_ErrorIdCmd.ERRORID_InvalidTargetSlot;
	ELSE
		//Vial in Slot ?
		pVial := pSlot^.P_pPiece;
		IF pVial = 0 THEN
			M_CheckAction := E_ErrorIdCmd.ERRORID_NoPieceInSlot;
		ELSE
			IF pVial^.P_eObjectType = E_ObjectType.OBJECTTYPE_VialClosed THEN
				M_CheckAction := E_ErrorIdCmd.ERRORID_InvalidPieceType;
			END_IF
		END_IF
	END_IF
ELSE
	M_CheckAction := SUPER^.M_CheckAction(refActionData, pCorrelObject);
END_IF
END_METHOD

METHOD M_GetAllProps : ERRORID
VAR_INPUT
	refCmdData : REFERENCE TO  ST_CmdData;
END_VAR
SUPER^.M_GetAllProps(refCmdData);
nCurrentPropIndex := nCurrentPropIndex + 1;
refCmdData.n32Data[nCurrentPropIndex] := nGCodeTargetNr;
END_METHOD

METHOD M_OverrideObjectType
VAR_INPUT
END_VAR
eObjectType := E_ObjectType.OBJECTTYPE_VialRackClosed;
END_METHOD

METHOD M_SetAllProps : ERRORID
VAR_INPUT
	refCmdData : REFERENCE TO  ST_CmdData;
END_VAR
M_SetAllProps := SUPER^.M_SetAllProps(refCmdData);

IF M_SetAllProps > 0 THEN
	RETURN;
END_IF

nCurrentPropIndex := nCurrentPropIndex + 1;
nGCodeTargetNr := DINT_TO_UINT(refCmdData.n32Data[nCurrentPropIndex]);
nNoOfProps := nCurrentPropIndex + 1;
END_METHOD

PROPERTY P_nGCodeTargetNr : UINT
GET
P_nGCodeTargetNr := nGCodeTargetNr;
END_GET
END_PROPERTY

END_FUNCTION_BLOCK

// ---- Objects/Pieces/FB_Vial.TcPOU
{attribute 'enable_dynamic_creation'}
FUNCTION_BLOCK FB_Vial EXTENDS FB_UsingPiece
VAR
	pSeptum: POINTER TO FB_PieceBase;
	nTopLevel: DINT;
	nBottomLevel: DINT;
END_VAR

{attribute 'object_name' := 'FB_init'}
METHOD FB_init : BOOL
VAR_INPUT
	/// if TRUE, the retain variables are initialized (warm start / cold start)
	bInitRetains: BOOL;
	/// if TRUE, the instance afterwards gets moved into the copy code (online change)
	bInCopyCode: BOOL;
END_VAR
bUsingPiece := TRUE;
eObjectType := E_ObjectType.OBJECTTYPE_Vial;
eObjectGroup := E_ObjectGroup.OBJECTGROUP_Piece;
END_METHOD

{attribute 'object_name' := 'M_ClearAllProps'}
METHOD M_ClearAllProps

VAR_INPUT
	bIgnoreParent : BOOL; //Es wird das gesamte OD gelöscht. -> Zeiger auf Parent nicht mehr gültig!
END_VAR
pSeptum := 0;
SUPER^.M_ClearAllProps(bIgnoreParent);
END_METHOD

{attribute 'object_name' := 'M_GetAllProps'}
METHOD M_GetAllProps : ERRORID
VAR_INPUT
	refCmdData: REFERENCE TO ST_CmdData;
END_VAR
SUPER^.M_GetAllProps(refCmdData);
nCurrentPropIndex := nCurrentPropIndex + 1;
refCmdData.n32Data[nCurrentPropIndex] := nTopLevel;
nCurrentPropIndex := nCurrentPropIndex + 1;
refCmdData.n32Data[nCurrentPropIndex] := nBottomLevel;
END_METHOD

{attribute 'object_name' := 'M_SetAllProps'}
METHOD M_SetAllProps : ERRORID
VAR_INPUT
	refCmdData: REFERENCE TO ST_CmdData;
END_VAR
M_SetAllProps := SUPER^.M_SetAllProps(refCmdData);

IF M_SetAllProps > 0 THEN
	RETURN;
END_IF
nCurrentPropIndex := nCurrentPropIndex + 1;
nTopLevel := refCmdData.n32Data[nCurrentPropIndex];
nCurrentPropIndex := nCurrentPropIndex + 1;
nBottomLevel := refCmdData.n32Data[nCurrentPropIndex];
nNoOfProps := nCurrentPropIndex + 1;
END_METHOD

METHOD M_SetSingleProp : ERRORID
VAR_INPUT
	refCmdData : REFERENCE TO  ST_CmdData;
END_VAR
IF refCmdData.aHeader[1] < 13 THEN	//Property-Nr
	M_SetSingleProp := SUPER^.M_SetSingleProp(refCmdData);
ELSE
	IF refCmdData.aHeader[1] = 13 THEN
		//bIsOpen := DINT_TO_BOOL(refCmdData.n32Data[0]);
		;
	ELSIF refCmdData.aHeader[1] = 14 THEN
		nTopLevel := refCmdData.n32Data[0];
	ELSIF refCmdData.aHeader[1] = 15 THEN
		nBottomLevel := refCmdData.n32Data[0];
	ELSE
		M_SetSingleProp := E_ErrorIdCmd.ERRORID_InvalidProperty;
	END_IF
END_IF
END_METHOD

PROPERTY P_nBottomLevel : DINT
GET
P_nBottomLevel := nBottomLevel;
END_GET
END_PROPERTY

PROPERTY P_nTopLevel : DINT
GET
P_nTopLevel := nTopLevel;
END_GET
END_PROPERTY

PROPERTY P_pLatestChild : POINTER TO FB_PieceBase
GET
IF pSeptum > 0 THEN
	P_pLatestChild := pSeptum;	
ELSE
	P_pLatestChild := THIS;
END_IF
END_GET
END_PROPERTY

PROPERTY P_pSeptum : POINTER TO FB_PieceBase
GET
P_pSeptum := pSeptum;
END_GET
SET
pSeptum := P_pSeptum;
END_SET
END_PROPERTY

END_FUNCTION_BLOCK

// ---- Sequence/FB_Sequence.TcPOU
{attribute 'enable_dynamic_creation'}
FUNCTION_BLOCK FB_Sequence
VAR_INPUT
END_VAR
VAR_OUTPUT
	eCurrentState	: E_SequenceState;
END_VAR
VAR
	nId					: UDINT;
	fbStepList			: FB_StepList();
	fbProcessingQueue 	: FB_ProcessingQueue;
	nMonitorStepNr		: UINT := 1;
	nMonitorStep 		: POINTER TO ST_Step;
	
	i					: UINT;
	pStep				: POINTER TO ST_Step;
	pFollowStep			: POINTER TO ST_Step;
	pLastStep			: POINTER TO ST_Step;
	
	bError				: BOOL;
	stError				: ST_Error;
	
	eOldState			: E_SequenceState;
	
	nCondiCheckResult	: BYTE; //Bit0 und Bit1 werden einzeln ausgewertet
	
	nCancelState		: USINT;
	
	nStepsReady			: UINT;
	
	eActionStatus		: E_ActionStatus;
	nInfo				: DINT;
	
	nSequParam			: UINT;
	nCounter			: DINT;
END_VAR

nMonitorStep := fbStepList.M_Get(nMonitorStepNr);	
//Sequence ruft den ActionDispacher auch, wie sonst FB_Auto
//auch die Untersequenzen werden von hier aufgerufen
stError.POUState := eCurrentState;

IF eOldState <> eCurrentState THEN
	fbSequenceInfo.M_AddTail(nId,eCurrentState,0);
	eOldState := eCurrentState;
END_IF

CASE eCurrentState OF
	E_SequenceState.State_Start:
		//InitialStep(1) und die Steps, welche keinen Forerunner haben in die ProcessingQueue eintragen
		fbProcessingQueue.M_Reset();
		nCancelState := 0;
		FOR i:= 1 TO fbStepList.P_nCount BY 1 DO	//Alle Steps durchlaufen
			pStep := fbStepList.M_Get(i);
			IF pStep > 0 THEN
				M_ChangeStepState(pStep,E_StepState.STEPSTATUS_Idle);
				M_ChangeStepInfo(pStep,0);
				pStep^.bFollowerInQueue := FALSE;
				IF NOT pStep^.bHasForerunner THEN
					fbProcessingQueue.M_Add(pStep);
					M_ChangeStepState(pStep,E_StepState.STEPSTATUS_InQueue);
				END_IF
			ELSE //Dieser Fall dürfte normalerweise nicht eintreten
				bError := TRUE;
				EXIT;
			END_IF
			//fbSequenceInfo.M_AddTail(nId,eCurrentState,pStep);
			//Auskommentiert, da bei sehr vielen Steps es zu Zyklusüberschreitungen kommen kann.
		END_FOR
		pLastStep := fbStepList.M_GetLast();
		fbComplexAction.P_nDispenseTrials := 0;
		eCurrentState := E_SequenceState.State_Active;
		
